LIN {X 0,Y 488.63,Z 370.241,A -85,B 0,C 180,E1 -6427.164,E2 -6427.164} C_VEL
LIN {X 0,Y 488.671,Z 370.238,A -85,B 0,C 180,E1 -6430.331,E2 -6430.331} C_VEL
LIN {X 0,Y 488.668,Z 370.24,A -85,B 0,C 180,E1 -6433.658,E2 -6433.658} C_VEL
LIN {X 0,Y 488.668,Z 370.231,A -85,B 0,C 180,E1 -6436.343,E2 -6436.343} C_VEL
LIN {X 0,Y 488.671,Z 370.225,A -85,B 0,C 180,E1 -6439.67,E2 -6439.67} C_VEL
LIN {X 0,Y 488.65,Z 370.243,A -85,B 0,C 180,E1 -6442.838,E2 -6442.838} C_VEL
LIN {X 0,Y 488.712,Z 370.223,A -85,B 0,C 180,E1 -6445.886,E2 -6445.886} C_VEL
LIN {X 0,Y 488.67,Z 370.24,A -85,B 0,C 180,E1 -6448.819,E2 -6448.819} C_VEL
LIN {X 0,Y 488.695,Z 370.235,A -85,B 0,C 180,E1 -6451.668,E2 -6451.668} C_VEL
LIN {X 0,Y 488.696,Z 370.239,A -85,B 0,C 180,E1 -6454.961,E2 -6454.961} C_VEL
LIN {X 0,Y 488.73,Z 370.261,A -85,B 0,C 180,E1 -6458.266,E2 -6458.266} C_VEL
LIN {X 0,Y 488.873,Z 371.046,A -85,B 0,C 180,E1 -6458.495,E2 -6458.495} C_VEL
LIN {X 0,Y 490.534,Z 379.437,A -85,B 0,C 180,E1 -6460.106,E2 -6460.106} C_VEL
LIN {X 0,Y 490.725,Z 380.846,A -85,B 0,C 180,E1 -6460.313,E2 -6460.313} C_VEL
LIN {X 0,Y 493.718,Z 393.755,A -85,B 0,C 180,E1 -6460.688,E2 -6460.688} C_VEL
LIN {X 0,Y 492.308,Z 519.715,A -85,B 0,C 180,E1 -6462.74,E2 -6462.74} C_VEL
LIN {X 0,Y 492.144,Z 534.173,A -85,B 0,C 180,E1 -6463.145,E2 -6463.145} C_VEL
LIN {X 0,Y 491.844,Z 548.393,A -85,B 0,C 180,E1 -6463.714,E2 -6463.714} C_VEL
LIN {X 0,Y 491.476,Z 562.149,A -85,B 0,C 180,E1 -6464.447,E2 -6464.447} C_VEL
LIN {X 0,Y 491.039,Z 573.092,A -85,B 0,C 180,E1 -6465.177,E2 -6465.177} C_VEL
LIN {X 0,Y 490.649,Z 584.683,A -85,B 0,C 180,E1 -6466.118,E2 -6466.118} C_VEL
LIN {X 0,Y 490.188,Z 595.699,A -85,B 0,C 180,E1 -6467.2,E2 -6467.2} C_VEL
LIN {X 0,Y 489.755,Z 605.882,A -85,B 0,C 180,E1 -6468.41,E2 -6468.41} C_VEL
LIN {X 0,Y 489.407,Z 614.564,A -85,B 0,C 180,E1 -6469.659,E2 -6469.659} C_VEL
LIN {X 0,Y 489.107,Z 622.847,A -85,B 0,C 180,E1 -6471.114,E2 -6471.114} C_VEL
LIN {X 0,Y 488.854,Z 629.502,A -85,B 0,C 180,E1 -6472.566,E2 -6472.566} C_VEL
LIN {X 0,Y 488.751,Z 634.11,A -85,B 0,C 180,E1 -6473.809,E2 -6473.809} C_VEL
LIN {X 0,Y 488.529,Z 637.769,A -85,B 0,C 180,E1 -6475.048,E2 -6475.048} C_VEL
LIN {X 0,Y 488.435,Z 641.375,A -85,B 0,C 180,E1 -6476.7,E2 -6476.7} C_VEL
LIN {X 0,Y 488.484,Z 642.64,A -85,B 0,C 180,E1 -6477.526,E2 -6477.526} C_VEL
LIN {X 0,Y 488.439,Z 644.177,A -85,B 0,C 180,E1 -6479.175,E2 -6479.175} C_VEL
LIN {X 0,Y 488.439,Z 644.37,A -85,B 0,C 180,E1 -6480.824,E2 -6480.824} C_VEL
LIN {X 0,Y 488.495,Z 643.209,A -85,B 0,C 180,E1 -6482.474,E2 -6482.474} C_VEL
LIN {X 0,Y 488.571,Z 640.686,A -85,B 0,C 180,E1 -6484.124,E2 -6484.124} C_VEL
LIN {X 0,Y 488.818,Z 636.708,A -85,B 0,C 180,E1 -6485.776,E2 -6485.776} C_VEL
LIN {X 0,Y 488.963,Z 631.462,A -85,B 0,C 180,E1 -6487.358,E2 -6487.358} C_VEL
LIN {X 0,Y 489.212,Z 625.844,A -85,B 0,C 180,E1 -6488.676,E2 -6488.676} C_VEL
LIN {X 0,Y 489.556,Z 618.17,A -85,B 0,C 180,E1 -6490.129,E2 -6490.129} C_VEL
LIN {X 0,Y 489.943,Z 610.105,A -85,B 0,C 180,E1 -6491.375,E2 -6491.375} C_VEL
LIN {X 0,Y 490.435,Z 600.545,A -85,B 0,C 180,E1 -6492.598,E2 -6492.598} C_VEL
LIN {X 0,Y 490.886,Z 589.425,A -85,B 0,C 180,E1 -6493.77,E2 -6493.77} C_VEL
LIN {X 0,Y 491.245,Z 578.536,A -85,B 0,C 180,E1 -6494.711,E2 -6494.711} C_VEL
LIN {X 0,Y 491.631,Z 566.669,A -85,B 0,C 180,E1 -6495.547,E2 -6495.547} C_VEL
LIN {X 0,Y 492.064,Z 553.581,A -85,B 0,C 180,E1 -6496.278,E2 -6496.278} C_VEL
LIN {X 0,Y 492.329,Z 540.591,A -85,B 0,C 180,E1 -6496.839,E2 -6496.839} C_VEL
LIN {X 0,Y 492.464,Z 526.256,A -85,B 0,C 180,E1 -6497.285,E2 -6497.285} C_VEL
LIN {X 0,Y 492.743,Z 500.215,A -85,B 0,C 180,E1 -6497.777,E2 -6497.777} C_VEL
LIN {X 0,Y 494.504,Z 408.672,A -85,B 0,C 180,E1 -6499.431,E2 -6499.431} C_VEL
LIN {X 0,Y 494.741,Z 394.774,A -85,B 0,C 180,E1 -6499.698,E2 -6499.698} C_VEL
LIN {X 0,Y 492.574,Z 387.053,A -85,B 0,C 180,E1 -6499.998,E2 -6499.998} C_VEL
LIN {X 0,Y 492.44,Z 385.522,A -85,B 0,C 180,E1 -6500.248,E2 -6500.248} C_VEL
LIN {X 0,Y 490.543,Z 377.295,A -85,B 0,C 180,E1 -6502.091,E2 -6502.091} C_VEL
LIN {X 0,Y 488.703,Z 370.295,A -85,B 0,C 180,E1 -6503.773,E2 -6503.773} C_VEL
LIN {X 0,Y 488.797,Z 370.226,A -85,B 0,C 180,E1 -6506.943,E2 -6506.943} C_VEL
LIN {X 0,Y 488.714,Z 370.236,A -85,B 0,C 180,E1 -6510.362,E2 -6510.362} C_VEL
LIN {X 0,Y 488.739,Z 370.23,A -85,B 0,C 180,E1 -6513.484,E2 -6513.484} C_VEL
LIN {X 0,Y 488.678,Z 370.241,A -85,B 0,C 180,E1 -6516.353,E2 -6516.353} C_VEL
LIN {X 0,Y 488.704,Z 370.234,A -85,B 0,C 180,E1 -6519.254,E2 -6519.254} C_VEL
LIN {X 0,Y 488.691,Z 370.24,A -85,B 0,C 180,E1 -6522.525,E2 -6522.525} C_VEL
LIN {X 0,Y 488.705,Z 370.234,A -85,B 0,C 180,E1 -6525.197,E2 -6525.197} C_VEL
LIN {X 0,Y 488.67,Z 370.241,A -85,B 0,C 180,E1 -6528.579,E2 -6528.579} C_VEL
LIN {X 0,Y 488.691,Z 370.237,A -85,B 0,C 180,E1 -6530.949,E2 -6530.949} C_VEL
LIN {X 0,Y 488.648,Z 370.246,A -85,B 0,C 180,E1 -6533.864,E2 -6533.864} C_VEL
LIN {X 0,Y 488.728,Z 370.463,A -85,B 0,C 180,E1 -6536.421,E2 -6536.421} C_VEL
LIN {X 0,Y 491.601,Z 379.515,A -85,B 0,C 180,E1 -6537.795,E2 -6537.795} C_VEL
LIN {X 0,Y 494.839,Z 392.145,A -85,B 0,C 180,E1 -6539.486,E2 -6539.486} C_VEL
LIN {X 0,Y 494.763,Z 398.434,A -85,B 0,C 180,E1 -6540.186,E2 -6540.186} C_VEL
LIN {X 0,Y 493.252,Z 428.365,A -85,B 0,C 180,E1 -6543.331,E2 -6543.331} C_VEL
LIN {X 0,Y 492.07,Z 458.993,A -85,B 0,C 180,E1 -6546.426,E2 -6546.426} C_VEL
LIN {X 0,Y 491.847,Z 465.628,A -85,B 0,C 180,E1 -6547.056,E2 -6547.056} C_VEL
LIN {X 0,Y 494.886,Z 488.681,A -85,B 0,C 180,E1 -6547.594,E2 -6547.594} C_VEL
LIN {X 0,Y 493.486,Z 641.012,A -85,B 0,C 180,E1 -6549.877,E2 -6549.877} C_VEL
LIN {X 0,Y 493.144,Z 656.633,A -85,B 0,C 180,E1 -6550.281,E2 -6550.281} C_VEL
LIN {X 0,Y 492.657,Z 671.656,A -85,B 0,C 180,E1 -6550.845,E2 -6550.845} C_VEL
LIN {X 0,Y 492.069,Z 686.298,A -85,B 0,C 180,E1 -6551.578,E2 -6551.578} C_VEL
LIN {X 0,Y 491.4,Z 699.566,A -85,B 0,C 180,E1 -6552.413,E2 -6552.413} C_VEL
LIN {X 0,Y 490.815,Z 711.781,A -85,B 0,C 180,E1 -6553.357,E2 -6553.357} C_VEL
LIN {X 0,Y 490.13,Z 724.205,A -85,B 0,C 180,E1 -6554.509,E2 -6554.509} C_VEL
LIN {X 0,Y 489.566,Z 736.347,A -85,B 0,C 180,E1 -6555.874,E2 -6555.874} C_VEL
LIN {X 0,Y 489.04,Z 747.102,A -85,B 0,C 180,E1 -6557.339,E2 -6557.339} C_VEL
LIN {X 0,Y 488.679,Z 756.035,A -85,B 0,C 180,E1 -6558.804,E2 -6558.804} C_VEL
LIN {X 0,Y 488.334,Z 764.373,A -85,B 0,C 180,E1 -6560.472,E2 -6560.472} C_VEL
LIN {X 0,Y 488.155,Z 771.047,A -85,B 0,C 180,E1 -6562.138,E2 -6562.138} C_VEL
LIN {X 0,Y 488.079,Z 775.38,A -85,B 0,C 180,E1 -6563.489,E2 -6563.489} C_VEL
LIN {X 0,Y 487.987,Z 779.262,A -85,B 0,C 180,E1 -6565.042,E2 -6565.042} C_VEL
LIN {X 0,Y 488.007,Z 782.201,A -85,B 0,C 180,E1 -6566.696,E2 -6566.696} C_VEL
LIN {X 0,Y 487.941,Z 783.951,A -85,B 0,C 180,E1 -6568.348,E2 -6568.348} C_VEL
LIN {X 0,Y 487.89,Z 784.548,A -85,B 0,C 180,E1 -6569.999,E2 -6569.999} C_VEL
LIN {X 0,Y 487.94,Z 783.95,A -85,B 0,C 180,E1 -6571.649,E2 -6571.649} C_VEL
LIN {X 0,Y 488.012,Z 782.198,A -85,B 0,C 180,E1 -6573.301,E2 -6573.301} C_VEL
LIN {X 0,Y 487.981,Z 779.264,A -85,B 0,C 180,E1 -6574.956,E2 -6574.956} C_VEL
LIN {X 0,Y 488.038,Z 775.078,A -85,B 0,C 180,E1 -6576.614,E2 -6576.614} C_VEL
LIN {X 0,Y 488.197,Z 769.522,A -85,B 0,C 180,E1 -6578.276,E2 -6578.276} C_VEL
LIN {X 0,Y 488.368,Z 762.446,A -85,B 0,C 180,E1 -6579.943,E2 -6579.943} C_VEL
LIN {X 0,Y 488.711,Z 754.857,A -85,B 0,C 180,E1 -6581.403,E2 -6581.403} C_VEL
LIN {X 0,Y 489.079,Z 745.703,A -85,B 0,C 180,E1 -6582.868,E2 -6582.868} C_VEL
LIN {X 0,Y 489.529,Z 736.367,A -85,B 0,C 180,E1 -6584.125,E2 -6584.125} C_VEL
LIN {X 0,Y 490.102,Z 724.237,A -85,B 0,C 180,E1 -6585.489,E2 -6585.489} C_VEL
LIN {X 0,Y 490.84,Z 711.822,A -85,B 0,C 180,E1 -6586.639,E2 -6586.639} C_VEL
LIN {X 0,Y 491.394,Z 699.601,A -85,B 0,C 180,E1 -6587.584,E2 -6587.584} C_VEL
LIN {X 0,Y 491.997,Z 686.334,A -85,B 0,C 180,E1 -6588.422,E2 -6588.422} C_VEL
LIN {X 0,Y 492.632,Z 671.724,A -85,B 0,C 180,E1 -6589.153,E2 -6589.153} C_VEL
LIN {X 0,Y 493.115,Z 656.455,A -85,B 0,C 180,E1 -6589.727,E2 -6589.727} C_VEL
LIN {X 0,Y 493.476,Z 641.155,A -85,B 0,C 180,E1 -6590.121,E2 -6590.121} C_VEL
LIN {X 0,Y 494.854,Z 499.188,A -85,B 0,C 180,E1 -6592.285,E2 -6592.285} C_VEL
LIN {X 0,Y 494.849,Z 487.544,A -85,B 0,C 180,E1 -6592.477,E2 -6592.477} C_VEL
LIN {X 0,Y 492.247,Z 468.47,A -85,B 0,C 180,E1 -6592.933,E2 -6592.933} C_VEL
LIN {X 0,Y 493.504,Z 436.983,A -85,B 0,C 180,E1 -6596.083,E2 -6596.083} C_VEL
LIN {X 0,Y 494.721,Z 409.612,A -85,B 0,C 180,E1 -6598.88,E2 -6598.88} C_VEL
LIN {X 0,Y 495.442,Z 394.035,A -85,B 0,C 180,E1 -6600.497,E2 -6600.497} C_VEL
LIN {X 0,Y 491.474,Z 379.619,A -85,B 0,C 180,E1 -6602.288,E2 -6602.288} C_VEL
LIN {X 0,Y 488.735,Z 370.407,A -85,B 0,C 180,E1 -6603.512,E2 -6603.512} C_VEL
LIN {X 0,Y 488.639,Z 370.245,A -85,B 0,C 180,E1 -6606.348,E2 -6606.348} C_VEL
LIN {X 0,Y 488.676,Z 370.237,A -85,B 0,C 180,E1 -6609.254,E2 -6609.254} C_VEL
LIN {X 0,Y 488.655,Z 370.244,A -85,B 0,C 180,E1 -6612.527,E2 -6612.527} C_VEL
LIN {X 0,Y 488.685,Z 370.234,A -85,B 0,C 180,E1 -6615.196,E2 -6615.196} C_VEL
LIN {X 0,Y 488.647,Z 370.228,A -85,B 0,C 180,E1 -6618.578,E2 -6618.578} C_VEL
LIN {X 0,Y 488.674,Z 370.237,A -85,B 0,C 180,E1 -6620.949,E2 -6620.949} C_VEL
LIN {X 0,Y 488.631,Z 370.228,A -85,B 0,C 180,E1 -6623.864,E2 -6623.864} C_VEL
LIN {X 0,Y 488.695,Z 370.226,A -85,B 0,C 180,E1 -6626.519,E2 -6626.519} C_VEL
LIN {X 0,Y 488.703,Z 370.232,A -85,B 0,C 180,E1 -6629.779,E2 -6629.779} C_VEL
LIN {X 0,Y 488.684,Z 370.234,A -85,B 0,C 180,E1 -6633.077,E2 -6633.077} C_VEL
LIN {X 0,Y 488.653,Z 370.236,A -85,B 0,C 180,E1 -6636.253,E2 -6636.253} C_VEL
LIN {X 0,Y 488.731,Z 370.223,A -85,B 0,C 180,E1 -6639.175,E2 -6639.175} C_VEL
LIN {X 0,Y 488.73,Z 370.226,A -85,B 0,C 180,E1 -6641.632,E2 -6641.632} C_VEL
LIN {X 0,Y 488.73,Z 370.223,A -85,B 0,C 180,E1 -6644.999,E2 -6644.999} C_VEL
LIN {X 0,Y 488.787,Z 370.228,A -85,B 0,C 180,E1 -6648.387,E2 -6648.387} C_VEL
LIN {X 0,Y 488.741,Z 370.223,A -85,B 0,C 180,E1 -6651.732,E2 -6651.732} C_VEL
LIN {X 0,Y 488.787,Z 370.224,A -85,B 0,C 180,E1 -6654.224,E2 -6654.224} C_VEL
LIN {X 0,Y 488.93,Z 370.201,A -85,B 0,C 180,E1 -6657.529,E2 -6657.529} C_VEL
LIN {X 0,Y 488.895,Z 370.203,A -85,B 0,C 180,E1 -6660.824,E2 -6660.824} C_VEL
LIN {X 0,Y 488.929,Z 370.203,A -85,B 0,C 180,E1 -6662.472,E2 -6662.472} C_VEL
LIN {X 0,Y 488.817,Z 370.213,A -85,B 0,C 180,E1 -6665.776,E2 -6665.776} C_VEL
LIN {X 0,Y 488.757,Z 370.224,A -85,B 0,C 180,E1 -6668.267,E2 -6668.267} C_VEL
LIN {X 0,Y 488.787,Z 370.212,A -85,B 0,C 180,E1 -6671.613,E2 -6671.613} C_VEL
LIN {X 0,Y 488.74,Z 370.226,A -85,B 0,C 180,E1 -6675.001,E2 -6675.001} C_VEL
LIN {X 0,Y 488.73,Z 370.23,A -85,B 0,C 180,E1 -6678.443,E2 -6678.443} C_VEL
LIN {X 0,Y 488.692,Z 370.23,A -85,B 0,C 180,E1 -6681.072,E2 -6681.072} C_VEL
LIN {X 0,Y 488.653,Z 370.237,A -85,B 0,C 180,E1 -6683.748,E2 -6683.748} C_VEL
LIN {X 0,Y 488.681,Z 370.24,A -85,B 0,C 180,E1 -6686.922,E2 -6686.922} C_VEL
LIN {X 0,Y 488.683,Z 370.234,A -85,B 0,C 180,E1 -6690.222,E2 -6690.222} C_VEL
LIN {X 0,Y 488.697,Z 370.234,A -85,B 0,C 180,E1 -6693.481,E2 -6693.481} C_VEL
LIN {X 0,Y 488.655,Z 370.235,A -85,B 0,C 180,E1 -6696.353,E2 -6696.353} C_VEL
LIN {X 0,Y 488.674,Z 370.238,A -85,B 0,C 180,E1 -6699.257,E2 -6699.257} C_VEL
LIN {X 0,Y 488.654,Z 370.232,A -85,B 0,C 180,E1 -6701.596,E2 -6701.596} C_VEL
LIN {X 0,Y 488.684,Z 370.242,A -85,B 0,C 180,E1 -6704.805,E2 -6704.805} C_VEL
LIN {X 0,Y 488.637,Z 370.24,A -85,B 0,C 180,E1 -6707.471,E2 -6707.471} C_VEL
LIN {X 0,Y 488.694,Z 370.229,A -85,B 0,C 180,E1 -6709.675,E2 -6709.675} C_VEL
LIN {X 0,Y 488.641,Z 370.237,A -85,B 0,C 180,E1 -6712.84,E2 -6712.84} C_VEL
LIN {X 0,Y 488.726,Z 370.405,A -85,B 0,C 180,E1 -6715.64,E2 -6715.64} C_VEL
LIN {X 0,Y 494.002,Z 388.467,A -85,B 0,C 180,E1 -6718.007,E2 -6718.007} C_VEL
LIN {X 0,Y 495.447,Z 393.988,A -85,B 0,C 180,E1 -6718.704,E2 -6718.704} C_VEL
LIN {X 0,Y 494.7,Z 414.108,A -85,B 0,C 180,E1 -6720.883,E2 -6720.883} C_VEL
LIN {X 0,Y 493.899,Z 418.535,A -85,B 0,C 180,E1 -6721.327,E2 -6721.327} C_VEL
LIN {X 0,Y 487.94,Z 433.643,A -85,B 0,C 180,E1 -6722.661,E2 -6722.661} C_VEL
LIN {X 0,Y 487.139,Z 438.124,A -85,B 0,C 180,E1 -6723.107,E2 -6723.107} C_VEL
LIN {X 0,Y 486.163,Z 465.721,A -85,B 0,C 180,E1 -6726.003,E2 -6726.003} C_VEL
LIN {X 0,Y 486.002,Z 472.632,A -85,B 0,C 180,E1 -6726.667,E2 -6726.667} C_VEL
LIN {X 0,Y 489.058,Z 491.11,A -85,B 0,C 180,E1 -6727.121,E2 -6727.121} C_VEL
LIN {X 0,Y 487.462,Z 640.161,A -85,B 0,C 180,E1 -6729.386,E2 -6729.386} C_VEL
LIN {X 0,Y 487.095,Z 655.841,A -85,B 0,C 180,E1 -6729.784,E2 -6729.784} C_VEL
LIN {X 0,Y 486.549,Z 669.962,A -85,B 0,C 180,E1 -6730.3,E2 -6730.3} C_VEL
LIN {X 0,Y 485.868,Z 684.559,A -85,B 0,C 180,E1 -6731.008,E2 -6731.008} C_VEL
LIN {X 0,Y 485.181,Z 698.293,A -85,B 0,C 180,E1 -6731.856,E2 -6731.856} C_VEL
LIN {X 0,Y 484.446,Z 710.916,A -85,B 0,C 180,E1 -6732.809,E2 -6732.809} C_VEL
LIN {X 0,Y 483.726,Z 723.662,A -85,B 0,C 180,E1 -6733.977,E2 -6733.977} C_VEL
LIN {X 0,Y 483.079,Z 733.473,A -85,B 0,C 180,E1 -6735.036,E2 -6735.036} C_VEL
LIN {X 0,Y 482.501,Z 743.486,A -85,B 0,C 180,E1 -6736.31,E2 -6736.31} C_VEL
LIN {X 0,Y 481.985,Z 753.507,A -85,B 0,C 180,E1 -6737.835,E2 -6737.835} C_VEL
LIN {X 0,Y 481.598,Z 761.397,A -85,B 0,C 180,E1 -6739.278,E2 -6739.278} C_VEL
LIN {X 0,Y 481.241,Z 768.131,A -85,B 0,C 180,E1 -6740.757,E2 -6740.757} C_VEL
LIN {X 0,Y 481.014,Z 774.375,A -85,B 0,C 180,E1 -6742.445,E2 -6742.445} C_VEL
LIN {X 0,Y 480.917,Z 779.203,A -85,B 0,C 180,E1 -6744.13,E2 -6744.13} C_VEL
LIN {X 0,Y 480.796,Z 782.742,A -85,B 0,C 180,E1 -6745.81,E2 -6745.81} C_VEL
LIN {X 0,Y 480.799,Z 785.083,A -85,B 0,C 180,E1 -6747.488,E2 -6747.488} C_VEL
LIN {X 0,Y 480.757,Z 786.278,A -85,B 0,C 180,E1 -6749.164,E2 -6749.164} C_VEL
LIN {X 0,Y 480.757,Z 786.295,A -85,B 0,C 180,E1 -6750.839,E2 -6750.839} C_VEL
LIN {X 0,Y 480.8,Z 785.169,A -85,B 0,C 180,E1 -6752.515,E2 -6752.515} C_VEL
LIN {X 0,Y 480.796,Z 782.895,A -85,B 0,C 180,E1 -6754.193,E2 -6754.193} C_VEL
LIN {X 0,Y 480.9,Z 779.42,A -85,B 0,C 180,E1 -6755.873,E2 -6755.873} C_VEL
LIN {X 0,Y 481.01,Z 774.663,A -85,B 0,C 180,E1 -6757.557,E2 -6757.557} C_VEL
LIN {X 0,Y 481.226,Z 768.503,A -85,B 0,C 180,E1 -6759.246,E2 -6759.246} C_VEL
LIN {X 0,Y 481.629,Z 760.754,A -85,B 0,C 180,E1 -6760.936,E2 -6760.936} C_VEL
LIN {X 0,Y 482.003,Z 752.225,A -85,B 0,C 180,E1 -6762.463,E2 -6762.463} C_VEL
LIN {X 0,Y 482.569,Z 742.54,A -85,B 0,C 180,E1 -6763.905,E2 -6763.905} C_VEL
LIN {X 0,Y 483.144,Z 732.385,A -85,B 0,C 180,E1 -6765.18,E2 -6765.18} C_VEL
LIN {X 0,Y 483.874,Z 720.993,A -85,B 0,C 180,E1 -6766.381,E2 -6766.381} C_VEL
LIN {X 0,Y 484.608,Z 708.092,A -85,B 0,C 180,E1 -6767.514,E2 -6767.514} C_VEL
LIN {X 0,Y 485.393,Z 694.88,A -85,B 0,C 180,E1 -6768.466,E2 -6768.466} C_VEL
LIN {X 0,Y 486.061,Z 681.287,A -85,B 0,C 180,E1 -6769.261,E2 -6769.261} C_VEL
LIN {X 0,Y 486.681,Z 666.702,A -85,B 0,C 180,E1 -6769.927,E2 -6769.927} C_VEL
LIN {X 0,Y 487.203,Z 651.649,A -85,B 0,C 180,E1 -6770.435,E2 -6770.435} C_VEL
LIN {X 0,Y 487.565,Z 635.65,A -85,B 0,C 180,E1 -6770.789,E2 -6770.789} C_VEL
LIN {X 0,Y 489.071,Z 490.942,A -85,B 0,C 180,E1 -6772.972,E2 -6772.972} C_VEL
LIN {X 0,Y 485.975,Z 472.205,A -85,B 0,C 180,E1 -6773.448,E2 -6773.448} C_VEL
LIN {X 0,Y 486.713,Z 448.579,A -85,B 0,C 180,E1 -6775.872,E2 -6775.872} C_VEL
LIN {X 0,Y 487.808,Z 421.261,A -85,B 0,C 180,E1 -6778.812,E2 -6778.812} C_VEL
LIN {X 0,Y 488.856,Z 396.737,A -85,B 0,C 180,E1 -6781.487,E2 -6781.487} C_VEL
LIN {X 0,Y 485.329,Z 383.414,A -85,B 0,C 180,E1 -6783.202,E2 -6783.202} C_VEL
LIN {X 0,Y 481.629,Z 371.34,A -85,B 0,C 180,E1 -6784.829,E2 -6784.829} C_VEL
LIN {X 0,Y 481.587,Z 371.116,A -85,B 0,C 180,E1 -6786.617,E2 -6786.617} C_VEL
LIN {X 0,Y 481.632,Z 371.111,A -85,B 0,C 180,E1 -6789.342,E2 -6789.342} C_VEL
LIN {X 0,Y 481.612,Z 371.107,A -85,B 0,C 180,E1 -6792.166,E2 -6792.166} C_VEL
LIN {X 0,Y 481.654,Z 371.112,A -85,B 0,C 180,E1 -6794.459,E2 -6794.459} C_VEL
LIN {X 0,Y 481.612,Z 371.117,A -85,B 0,C 180,E1 -6797.835,E2 -6797.835} C_VEL
LIN {X 0,Y 481.625,Z 371.11,A -85,B 0,C 180,E1 -6801.136,E2 -6801.136} C_VEL
LIN {X 0,Y 481.618,Z 371.108,A -85,B 0,C 180,E1 -6804.289,E2 -6804.289} C_VEL
LIN {X 0,Y 481.675,Z 371.099,A -85,B 0,C 180,E1 -6806.327,E2 -6806.327} C_VEL
LIN {X 0,Y 481.631,Z 371.118,A -85,B 0,C 180,E1 -6809.423,E2 -6809.423} C_VEL
LIN {X 0,Y 481.649,Z 371.111,A -85,B 0,C 180,E1 -6812.165,E2 -6812.165} C_VEL
LIN {X 0,Y 481.67,Z 371.114,A -85,B 0,C 180,E1 -6814.967,E2 -6814.967} C_VEL
LIN {X 0,Y 481.708,Z 371.32,A -85,B 0,C 180,E1 -6818.13,E2 -6818.13} C_VEL
LIN {X 0,Y 483.601,Z 380.575,A -85,B 0,C 180,E1 -6819.919,E2 -6819.919} C_VEL
LIN {X 0,Y 483.905,Z 381.906,A -85,B 0,C 180,E1 -6820.05,E2 -6820.05} C_VEL
LIN {X 0,Y 486.909,Z 394.286,A -85,B 0,C 180,E1 -6820.41,E2 -6820.41} C_VEL
LIN {X 0,Y 485.9,Z 484.424,A -85,B 0,C 180,E1 -6821.909,E2 -6821.909} C_VEL
LIN {X 0,Y 485.496,Z 520.889,A -85,B 0,C 180,E1 -6822.528,E2 -6822.528} C_VEL
LIN {X 0,Y 485.33,Z 535.642,A -85,B 0,C 180,E1 -6822.955,E2 -6822.955} C_VEL
LIN {X 0,Y 485.008,Z 549.682,A -85,B 0,C 180,E1 -6823.532,E2 -6823.532} C_VEL
LIN {X 0,Y 484.641,Z 562.452,A -85,B 0,C 180,E1 -6824.222,E2 -6824.222} C_VEL
LIN {X 0,Y 484.2,Z 573.506,A -85,B 0,C 180,E1 -6824.963,E2 -6824.963} C_VEL
LIN {X 0,Y 483.779,Z 585.19,A -85,B 0,C 180,E1 -6825.917,E2 -6825.917} C_VEL
LIN {X 0,Y 483.275,Z 596.818,A -85,B 0,C 180,E1 -6827.071,E2 -6827.071} C_VEL
LIN {X 0,Y 482.838,Z 606.54,A -85,B 0,C 180,E1 -6828.242,E2 -6828.242} C_VEL
LIN {X 0,Y 482.462,Z 615.289,A -85,B 0,C 180,E1 -6829.509,E2 -6829.509} C_VEL
LIN {X 0,Y 482.127,Z 623.647,A -85,B 0,C 180,E1 -6830.984,E2 -6830.984} C_VEL
LIN {X 0,Y 481.875,Z 630.351,A -85,B 0,C 180,E1 -6832.457,E2 -6832.457} C_VEL
LIN {X 0,Y 481.76,Z 634.996,A -85,B 0,C 180,E1 -6833.719,E2 -6833.719} C_VEL
LIN {X 0,Y 481.496,Z 639.77,A -85,B 0,C 180,E1 -6835.395,E2 -6835.395} C_VEL
LIN {X 0,Y 481.412,Z 642.347,A -85,B 0,C 180,E1 -6836.652,E2 -6836.652} C_VEL
LIN {X 0,Y 481.471,Z 643.628,A -85,B 0,C 180,E1 -6837.49,E2 -6837.49} C_VEL
LIN {X 0,Y 481.426,Z 645.196,A -85,B 0,C 180,E1 -6839.163,E2 -6839.163} C_VEL
LIN {X 0,Y 481.427,Z 645.413,A -85,B 0,C 180,E1 -6840.836,E2 -6840.836} C_VEL
LIN {X 0,Y 481.486,Z 644.266,A -85,B 0,C 180,E1 -6842.51,E2 -6842.51} C_VEL
LIN {X 0,Y 481.567,Z 641.75,A -85,B 0,C 180,E1 -6844.185,E2 -6844.185} C_VEL
LIN {X 0,Y 481.836,Z 637.77,A -85,B 0,C 180,E1 -6845.86,E2 -6845.86} C_VEL
LIN {X 0,Y 481.995,Z 632.523,A -85,B 0,C 180,E1 -6847.467,E2 -6847.467} C_VEL
LIN {X 0,Y 482.27,Z 626.922,A -85,B 0,C 180,E1 -6848.802,E2 -6848.802} C_VEL
LIN {X 0,Y 482.66,Z 619.262,A -85,B 0,C 180,E1 -6850.275,E2 -6850.275} C_VEL
LIN {X 0,Y 483.085,Z 611.189,A -85,B 0,C 180,E1 -6851.539,E2 -6851.539} C_VEL
LIN {X 0,Y 483.581,Z 601.61,A -85,B 0,C 180,E1 -6852.779,E2 -6852.779} C_VEL
LIN {X 0,Y 484.07,Z 590.454,A -85,B 0,C 180,E1 -6853.967,E2 -6853.967} C_VEL
LIN {X 0,Y 484.462,Z 579.527,A -85,B 0,C 180,E1 -6854.921,E2 -6854.921} C_VEL
LIN {X 0,Y 484.862,Z 567.644,A -85,B 0,C 180,E1 -6855.77,E2 -6855.77} C_VEL
LIN {X 0,Y 485.339,Z 554.6,A -85,B 0,C 180,E1 -6856.51,E2 -6856.51} C_VEL
LIN {X 0,Y 485.61,Z 542.435,A -85,B 0,C 180,E1 -6857.051,E2 -6857.051} C_VEL
LIN {X 0,Y 485.715,Z 528.411,A -85,B 0,C 180,E1 -6857.51,E2 -6857.51} C_VEL
LIN {X 0,Y 485.959,Z 507.762,A -85,B 0,C 180,E1 -6857.925,E2 -6857.925} C_VEL
LIN {X 0,Y 487.743,Z 420.488,A -85,B 0,C 180,E1 -6859.546,E2 -6859.546} C_VEL
LIN {X 0,Y 488.183,Z 395.696,A -85,B 0,C 180,E1 -6860.039,E2 -6860.039} C_VEL
LIN {X 0,Y 485.964,Z 388.277,A -85,B 0,C 180,E1 -6860.344,E2 -6860.344} C_VEL
LIN {X 0,Y 485.648,Z 387.025,A -85,B 0,C 180,E1 -6860.544,E2 -6860.544} C_VEL
LIN {X 0,Y 483.703,Z 378.84,A -85,B 0,C 180,E1 -6862.42,E2 -6862.42} C_VEL
LIN {X 0,Y 481.715,Z 371.165,A -85,B 0,C 180,E1 -6864.312,E2 -6864.312} C_VEL
LIN {X 0,Y 481.751,Z 371.104,A -85,B 0,C 180,E1 -6867.139,E2 -6867.139} C_VEL
LIN {X 0,Y 481.684,Z 371.11,A -85,B 0,C 180,E1 -6869.741,E2 -6869.741} C_VEL
LIN {X 0,Y 481.677,Z 371.113,A -85,B 0,C 180,E1 -6872.674,E2 -6872.674} C_VEL
LIN {X 0,Y 481.665,Z 371.112,A -85,B 0,C 180,E1 -6875.203,E2 -6875.203} C_VEL
LIN {X 0,Y 481.674,Z 371.112,A -85,B 0,C 180,E1 -6878.859,E2 -6878.859} C_VEL
LIN {X 0,Y 481.65,Z 371.116,A -85,B 0,C 180,E1 -6881.911,E2 -6881.911} C_VEL
LIN {X 0,Y 481.658,Z 371.116,A -85,B 0,C 180,E1 -6884.457,E2 -6884.457} C_VEL
LIN {X 0,Y 481.628,Z 371.119,A -85,B 0,C 180,E1 -6887.836,E2 -6887.836} C_VEL
LIN {X 0,Y 481.652,Z 371.115,A -85,B 0,C 180,E1 -6890.655,E2 -6890.655} C_VEL
LIN {X 0,Y 481.609,Z 371.119,A -85,B 0,C 180,E1 -6893.379,E2 -6893.379} C_VEL
LIN {X 0,Y 481.708,Z 371.307,A -85,B 0,C 180,E1 -6895.905,E2 -6895.905} C_VEL
LIN {X 0,Y 485.064,Z 381.911,A -85,B 0,C 180,E1 -6897.581,E2 -6897.581} C_VEL
LIN {X 0,Y 488.184,Z 394.044,A -85,B 0,C 180,E1 -6899.265,E2 -6899.265} C_VEL
LIN {X 0,Y 488.26,Z 398.178,A -85,B 0,C 180,E1 -6899.748,E2 -6899.748} C_VEL
LIN {X 0,Y 486.737,Z 424.588,A -85,B 0,C 180,E1 -6902.596,E2 -6902.596} C_VEL
LIN {X 0,Y 485.382,Z 455.536,A -85,B 0,C 180,E1 -6905.811,E2 -6905.811} C_VEL
LIN {X 0,Y 485.056,Z 464.405,A -85,B 0,C 180,E1 -6906.687,E2 -6906.687} C_VEL
LIN {X 0,Y 486.937,Z 479.661,A -85,B 0,C 180,E1 -6907.064,E2 -6907.064} C_VEL
LIN {X 0,Y 488.303,Z 490.714,A -85,B 0,C 180,E1 -6907.304,E2 -6907.304} C_VEL
LIN {X 0,Y 486.839,Z 641.179,A -85,B 0,C 180,E1 -6909.59,E2 -6909.59} C_VEL
LIN {X 0,Y 486.468,Z 656.504,A -85,B 0,C 180,E1 -6909.991,E2 -6909.991} C_VEL
LIN {X 0,Y 485.957,Z 671.728,A -85,B 0,C 180,E1 -6910.57,E2 -6910.57} C_VEL
LIN {X 0,Y 485.293,Z 686.354,A -85,B 0,C 180,E1 -6911.311,E2 -6911.311} C_VEL
LIN {X 0,Y 484.633,Z 699.612,A -85,B 0,C 180,E1 -6912.16,E2 -6912.16} C_VEL
LIN {X 0,Y 483.922,Z 712.988,A -85,B 0,C 180,E1 -6913.215,E2 -6913.215} C_VEL
LIN {X 0,Y 483.179,Z 725.264,A -85,B 0,C 180,E1 -6914.389,E2 -6914.389} C_VEL
LIN {X 0,Y 482.628,Z 736.375,A -85,B 0,C 180,E1 -6915.666,E2 -6915.666} C_VEL
LIN {X 0,Y 482.051,Z 747.126,A -85,B 0,C 180,E1 -6917.153,E2 -6917.153} C_VEL
LIN {X 0,Y 481.67,Z 756.056,A -85,B 0,C 180,E1 -6918.639,E2 -6918.639} C_VEL
LIN {X 0,Y 481.27,Z 764.392,A -85,B 0,C 180,E1 -6920.331,E2 -6920.331} C_VEL
LIN {X 0,Y 481.105,Z 771.064,A -85,B 0,C 180,E1 -6922.022,E2 -6922.022} C_VEL
LIN {X 0,Y 481.007,Z 775.675,A -85,B 0,C 180,E1 -6923.488,E2 -6923.488} C_VEL
LIN {X 0,Y 480.913,Z 779.277,A -85,B 0,C 180,E1 -6924.968,E2 -6924.968} C_VEL
LIN {X 0,Y 480.931,Z 782.215,A -85,B 0,C 180,E1 -6926.648,E2 -6926.648} C_VEL
LIN {X 0,Y 480.869,Z 783.965,A -85,B 0,C 180,E1 -6928.324,E2 -6928.324} C_VEL
LIN {X 0,Y 480.809,Z 784.562,A -85,B 0,C 180,E1 -6929.999,E2 -6929.999} C_VEL
LIN {X 0,Y 480.868,Z 783.964,A -85,B 0,C 180,E1 -6931.674,E2 -6931.674} C_VEL
LIN {X 0,Y 480.934,Z 782.213,A -85,B 0,C 180,E1 -6933.35,E2 -6933.35} C_VEL
LIN {X 0,Y 480.906,Z 779.28,A -85,B 0,C 180,E1 -6935.029,E2 -6935.029} C_VEL
LIN {X 0,Y 480.958,Z 775.094,A -85,B 0,C 180,E1 -6936.712,E2 -6936.712} C_VEL
LIN {X 0,Y 481.113,Z 769.539,A -85,B 0,C 180,E1 -6938.398,E2 -6938.398} C_VEL
LIN {X 0,Y 481.326,Z 762.465,A -85,B 0,C 180,E1 -6940.09,E2 -6940.09} C_VEL
LIN {X 0,Y 481.667,Z 754.879,A -85,B 0,C 180,E1 -6941.572,E2 -6941.572} C_VEL
LIN {X 0,Y 482.091,Z 745.728,A -85,B 0,C 180,E1 -6943.058,E2 -6943.058} C_VEL
LIN {X 0,Y 482.587,Z 736.394,A -85,B 0,C 180,E1 -6944.332,E2 -6944.332} C_VEL
LIN {X 0,Y 483.154,Z 725.293,A -85,B 0,C 180,E1 -6945.609,E2 -6945.609} C_VEL
LIN {X 0,Y 483.946,Z 713.078,A -85,B 0,C 180,E1 -6946.777,E2 -6946.777} C_VEL
LIN {X 0,Y 484.609,Z 699.647,A -85,B 0,C 180,E1 -6947.839,E2 -6947.839} C_VEL
LIN {X 0,Y 485.244,Z 686.389,A -85,B 0,C 180,E1 -6948.688,E2 -6948.688} C_VEL
LIN {X 0,Y 485.928,Z 671.793,A -85,B 0,C 180,E1 -6949.428,E2 -6949.428} C_VEL
LIN {X 0,Y 486.442,Z 656.797,A -85,B 0,C 180,E1 -6950.001,E2 -6950.001} C_VEL
LIN {X 0,Y 486.828,Z 641.309,A -85,B 0,C 180,E1 -6950.408,E2 -6950.408} C_VEL
LIN {X 0,Y 488.314,Z 489.212,A -85,B 0,C 180,E1 -6952.738,E2 -6952.738} C_VEL
LIN {X 0,Y 485.405,Z 467.989,A -85,B 0,C 180,E1 -6953.25,E2 -6953.25} C_VEL
LIN {X 0,Y 486.751,Z 437.596,A -85,B 0,C 180,E1 -6956.331,E2 -6956.331} C_VEL
LIN {X 0,Y 488.037,Z 409.988,A -85,B 0,C 180,E1 -6959.195,E2 -6959.195} C_VEL
LIN {X 0,Y 488.699,Z 395.715,A -85,B 0,C 180,E1 -6960.696,E2 -6960.696} C_VEL
LIN {X 0,Y 483.657,Z 377.985,A -85,B 0,C 180,E1 -6962.949,E2 -6962.949} C_VEL
LIN {X 0,Y 481.692,Z 371.271,A -85,B 0,C 180,E1 -6963.868,E2 -6963.868} C_VEL
LIN {X 0,Y 481.595,Z 371.12,A -85,B 0,C 180,E1 -6966.747,E2 -6966.747} C_VEL
LIN {X 0,Y 481.644,Z 371.116,A -85,B 0,C 180,E1 -6969.941,E2 -6969.941} C_VEL
LIN {X 0,Y 481.61,Z 371.115,A -85,B 0,C 180,E1 -6973.301,E2 -6973.301} C_VEL
LIN {X 0,Y 481.636,Z 371.113,A -85,B 0,C 180,E1 -6975.641,E2 -6975.641} C_VEL
LIN {X 0,Y 481.609,Z 371.11,A -85,B 0,C 180,E1 -6978.953,E2 -6978.953} C_VEL
LIN {X 0,Y 481.616,Z 371.118,A -85,B 0,C 180,E1 -6981.996,E2 -6981.996} C_VEL
LIN {X 0,Y 481.664,Z 371.089,A -85,B 0,C 180,E1 -6985.316,E2 -6985.316} C_VEL
LIN {X 0,Y 481.627,Z 371.118,A -85,B 0,C 180,E1 -6988.31,E2 -6988.31} C_VEL
LIN {X 0,Y 481.644,Z 371.107,A -85,B 0,C 180,E1 -6991.215,E2 -6991.215} C_VEL
LIN {X 0,Y 481.63,Z 371.115,A -85,B 0,C 180,E1 -6994.039,E2 -6994.039} C_VEL
LIN {X 0,Y 481.638,Z 371.115,A -85,B 0,C 180,E1 -6996.817,E2 -6996.817} C_VEL
LIN {X 0,Y 481.676,Z 371.101,A -85,B 0,C 180,E1 -6999.502,E2 -6999.502} C_VEL
LIN {X 0,Y 481.652,Z 371.112,A -85,B 0,C 180,E1 -7002.156,E2 -7002.156} C_VEL
LIN {X 0,Y 481.712,Z 371.098,A -85,B 0,C 180,E1 -7004.775,E2 -7004.775} C_VEL
LIN {X 0,Y 481.733,Z 371.104,A -85,B 0,C 180,E1 -7008.215,E2 -7008.215} C_VEL
LIN {X 0,Y 481.7,Z 371.099,A -85,B 0,C 180,E1 -7011.611,E2 -7011.611} C_VEL
LIN {X 0,Y 481.748,Z 371.1,A -85,B 0,C 180,E1 -7014.139,E2 -7014.139} C_VEL
LIN {X 0,Y 481.897,Z 371.077,A -85,B 0,C 180,E1 -7017.492,E2 -7017.492} C_VEL
LIN {X 0,Y 481.848,Z 371.08,A -85,B 0,C 180,E1 -7020.836,E2 -7020.836} C_VEL
LIN {X 0,Y 481.895,Z 371.079,A -85,B 0,C 180,E1 -7022.508,E2 -7022.508} C_VEL
LIN {X 0,Y 481.777,Z 371.091,A -85,B 0,C 180,E1 -7025.861,E2 -7025.861} C_VEL
LIN {X 0,Y 481.712,Z 371.103,A -85,B 0,C 180,E1 -7028.389,E2 -7028.389} C_VEL
LIN {X 0,Y 481.733,Z 371.09,A -85,B 0,C 180,E1 -7031.785,E2 -7031.785} C_VEL
LIN {X 0,Y 481.723,Z 371.098,A -85,B 0,C 180,E1 -7035.225,E2 -7035.225} C_VEL
LIN {X 0,Y 481.692,Z 371.111,A -85,B 0,C 180,E1 -7038.723,E2 -7038.723} C_VEL
LIN {X 0,Y 481.63,Z 371.108,A -85,B 0,C 180,E1 -7041.396,E2 -7041.396} C_VEL
LIN {X 0,Y 481.632,Z 371.114,A -85,B 0,C 180,E1 -7044.116,E2 -7044.116} C_VEL
LIN {X 0,Y 481.636,Z 371.115,A -85,B 0,C 180,E1 -7047.118,E2 -7047.118} C_VEL
LIN {X 0,Y 481.637,Z 371.109,A -85,B 0,C 180,E1 -7049.744,E2 -7049.744} C_VEL
LIN {X 0,Y 481.635,Z 371.115,A -85,B 0,C 180,E1 -7052.677,E2 -7052.677} C_VEL
LIN {X 0,Y 481.616,Z 371.113,A -85,B 0,C 180,E1 -7055.711,E2 -7055.711} C_VEL
LIN {X 0,Y 481.618,Z 371.111,A -85,B 0,C 180,E1 -7058.864,E2 -7058.864} C_VEL
LIN {X 0,Y 481.608,Z 371.109,A -85,B 0,C 180,E1 -7061.91,E2 -7061.91} C_VEL
LIN {X 0,Y 481.638,Z 371.115,A -85,B 0,C 180,E1 -7064.46,E2 -7064.46} C_VEL
LIN {X 0,Y 481.601,Z 371.111,A -85,B 0,C 180,E1 -7066.857,E2 -7066.857} C_VEL
LIN {X 0,Y 481.645,Z 371.106,A -85,B 0,C 180,E1 -7070.059,E2 -7070.059} C_VEL
LIN {X 0,Y 481.599,Z 371.114,A -85,B 0,C 180,E1 -7073.381,E2 -7073.381} C_VEL
LIN {X 0,Y 481.678,Z 371.192,A -85,B 0,C 180,E1 -7075.223,E2 -7075.223} C_VEL
LIN {X 0,Y 481.976,Z 372.457,A -85,B 0,C 180,E1 -7075.447,E2 -7075.447} C_VEL
LIN {X 0,Y 486.926,Z 389.013,A -85,B 0,C 180,E1 -7077.626,E2 -7077.626} C_VEL
LIN {X 0,Y 488.808,Z 396.09,A -85,B 0,C 180,E1 -7078.531,E2 -7078.531} C_VEL
LIN {X 0,Y 487.944,Z 416.867,A -85,B 0,C 180,E1 -7080.799,E2 -7080.799} C_VEL
LIN {X 0,Y 487.139,Z 438.124,A -85,B 0,C 180,E1 -7083.107,E2 -7083.107} C_VEL
LIN {X 0,Y 486.343,Z 442.609,A -85,B 0,C 180,E1 -7083.55,E2 -7083.55} C_VEL
LIN {X 0,Y 480.372,Z 457.882,A -85,B 0,C 180,E1 -7084.878,E2 -7084.878} C_VEL
LIN {X 0,Y 479.565,Z 462.435,A -85,B 0,C 180,E1 -7085.32,E2 -7085.32} C_VEL
LIN {X 0,Y 479.316,Z 472.55,A -85,B 0,C 180,E1 -7086.322,E2 -7086.322} C_VEL
LIN {X 0,Y 482.522,Z 492.251,A -85,B 0,C 180,E1 -7086.813,E2 -7086.813} C_VEL
LIN {X 0,Y 480.811,Z 640.401,A -85,B 0,C 180,E1 -7089.095,E2 -7089.095} C_VEL
LIN {X 0,Y 480.411,Z 656.314,A -85,B 0,C 180,E1 -7089.508,E2 -7089.508} C_VEL
LIN {X 0,Y 479.854,Z 670.237,A -85,B 0,C 180,E1 -7090.029,E2 -7090.029} C_VEL
LIN {X 0,Y 479.144,Z 684.518,A -85,B 0,C 180,E1 -7090.731,E2 -7090.731} C_VEL
LIN {X 0,Y 478.399,Z 698.258,A -85,B 0,C 180,E1 -7091.59,E2 -7091.59} C_VEL
LIN {X 0,Y 477.635,Z 710.885,A -85,B 0,C 180,E1 -7092.556,E2 -7092.556} C_VEL
LIN {X 0,Y 476.862,Z 723.636,A -85,B 0,C 180,E1 -7093.74,E2 -7093.74} C_VEL
LIN {X 0,Y 476.065,Z 735.197,A -85,B 0,C 180,E1 -7095.03,E2 -7095.03} C_VEL
LIN {X 0,Y 475.422,Z 744.943,A -85,B 0,C 180,E1 -7096.32,E2 -7096.32} C_VEL
LIN {X 0,Y 474.955,Z 754.014,A -85,B 0,C 180,E1 -7097.746,E2 -7097.746} C_VEL
LIN {X 0,Y 474.505,Z 762.423,A -85,B 0,C 180,E1 -7099.332,E2 -7099.332} C_VEL
LIN {X 0,Y 474.109,Z 769.832,A -85,B 0,C 180,E1 -7101.047,E2 -7101.047} C_VEL
LIN {X 0,Y 473.908,Z 775.717,A -85,B 0,C 180,E1 -7102.76,E2 -7102.76} C_VEL
LIN {X 0,Y 473.82,Z 779.189,A -85,B 0,C 180,E1 -7104.042,E2 -7104.042} C_VEL
LIN {X 0,Y 473.705,Z 782.728,A -85,B 0,C 180,E1 -7105.747,E2 -7105.747} C_VEL
LIN {X 0,Y 473.718,Z 785.069,A -85,B 0,C 180,E1 -7107.45,E2 -7107.45} C_VEL
LIN {X 0,Y 473.685,Z 786.264,A -85,B 0,C 180,E1 -7109.151,E2 -7109.151} C_VEL
LIN {X 0,Y 473.686,Z 786.281,A -85,B 0,C 180,E1 -7110.851,E2 -7110.851} C_VEL
LIN {X 0,Y 473.719,Z 785.155,A -85,B 0,C 180,E1 -7112.552,E2 -7112.552} C_VEL
LIN {X 0,Y 473.705,Z 782.879,A -85,B 0,C 180,E1 -7114.255,E2 -7114.255} C_VEL
LIN {X 0,Y 473.816,Z 779.402,A -85,B 0,C 180,E1 -7115.961,E2 -7115.961} C_VEL
LIN {X 0,Y 473.951,Z 774.643,A -85,B 0,C 180,E1 -7117.671,E2 -7117.671} C_VEL
LIN {X 0,Y 474.183,Z 768.481,A -85,B 0,C 180,E1 -7119.384,E2 -7119.384} C_VEL
LIN {X 0,Y 474.612,Z 760.73,A -85,B 0,C 180,E1 -7121.1,E2 -7121.1} C_VEL
LIN {X 0,Y 475.002,Z 752.474,A -85,B 0,C 180,E1 -7122.605,E2 -7122.605} C_VEL
LIN {X 0,Y 475.627,Z 742.508,A -85,B 0,C 180,E1 -7124.113,E2 -7124.113} C_VEL
LIN {X 0,Y 476.229,Z 732.348,A -85,B 0,C 180,E1 -7125.406,E2 -7125.406} C_VEL
LIN {X 0,Y 476.983,Z 720.952,A -85,B 0,C 180,E1 -7126.625,E2 -7126.625} C_VEL
LIN {X 0,Y 477.812,Z 708.046,A -85,B 0,C 180,E1 -7127.772,E2 -7127.772} C_VEL
LIN {X 0,Y 478.615,Z 694.826,A -85,B 0,C 180,E1 -7128.737,E2 -7128.737} C_VEL
LIN {X 0,Y 479.349,Z 681.223,A -85,B 0,C 180,E1 -7129.541,E2 -7129.541} C_VEL
LIN {X 0,Y 480.008,Z 666.319,A -85,B 0,C 180,E1 -7130.229,E2 -7130.229} C_VEL
LIN {X 0,Y 480.598,Z 651.01,A -85,B 0,C 180,E1 -7130.743,E2 -7130.743} C_VEL
LIN {X 0,Y 480.926,Z 635.279,A -85,B 0,C 180,E1 -7131.092,E2 -7131.092} C_VEL
LIN {X 0,Y 482.479,Z 491.439,A -85,B 0,C 180,E1 -7133.293,E2 -7133.293} C_VEL
LIN {X 0,Y 479.29,Z 472.305,A -85,B 0,C 180,E1 -7133.782,E2 -7133.782} C_VEL
LIN {X 0,Y 479.887,Z 452.379,A -85,B 0,C 180,E1 -7135.83,E2 -7135.83} C_VEL
LIN {X 0,Y 481.084,Z 424.672,A -85,B 0,C 180,E1 -7138.823,E2 -7138.823} C_VEL
LIN {X 0,Y 482.226,Z 399.029,A -85,B 0,C 180,E1 -7141.647,E2 -7141.647} C_VEL
LIN {X 0,Y 479.32,Z 387.781,A -85,B 0,C 180,E1 -7143.109,E2 -7143.109} C_VEL
LIN {X 0,Y 474.576,Z 372.176,A -85,B 0,C 180,E1 -7145.237,E2 -7145.237} C_VEL
LIN {X 0,Y 474.583,Z 371.991,A -85,B 0,C 180,E1 -7148.461,E2 -7148.461} C_VEL
LIN {X 0,Y 474.583,Z 371.983,A -85,B 0,C 180,E1 -7151.791,E2 -7151.791} C_VEL
LIN {X 0,Y 474.613,Z 371.988,A -85,B 0,C 180,E1 -7154.702,E2 -7154.702} C_VEL
LIN {X 0,Y 474.584,Z 371.991,A -85,B 0,C 180,E1 -7158.211,E2 -7158.211} C_VEL
LIN {X 0,Y 474.587,Z 371.994,A -85,B 0,C 180,E1 -7161.54,E2 -7161.54} C_VEL
LIN {X 0,Y 474.613,Z 371.977,A -85,B 0,C 180,E1 -7164.725,E2 -7164.725} C_VEL
LIN {X 0,Y 474.614,Z 371.988,A -85,B 0,C 180,E1 -7167.786,E2 -7167.786} C_VEL
LIN {X 0,Y 474.597,Z 371.994,A -85,B 0,C 180,E1 -7170.892,E2 -7170.892} C_VEL
LIN {X 0,Y 474.575,Z 371.995,A -85,B 0,C 180,E1 -7173.623,E2 -7173.623} C_VEL
LIN {X 0,Y 474.638,Z 371.988,A -85,B 0,C 180,E1 -7176.642,E2 -7176.642} C_VEL
LIN {X 0,Y 474.64,Z 372.155,A -85,B 0,C 180,E1 -7177.873,E2 -7177.873} C_VEL
LIN {X 0,Y 476.711,Z 381.803,A -85,B 0,C 180,E1 -7179.722,E2 -7179.722} C_VEL
LIN {X 0,Y 479.069,Z 390.159,A -85,B 0,C 180,E1 -7179.995,E2 -7179.995} C_VEL
LIN {X 0,Y 480.339,Z 396.61,A -85,B 0,C 180,E1 -7180.166,E2 -7180.166} C_VEL
LIN {X 0,Y 478.705,Z 521.115,A -85,B 0,C 180,E1 -7182.289,E2 -7182.289} C_VEL
LIN {X 0,Y 478.53,Z 536.001,A -85,B 0,C 180,E1 -7182.721,E2 -7182.721} C_VEL
LIN {X 0,Y 478.215,Z 549.82,A -85,B 0,C 180,E1 -7183.292,E2 -7183.292} C_VEL
LIN {X 0,Y 477.833,Z 562.746,A -85,B 0,C 180,E1 -7183.992,E2 -7183.992} C_VEL
LIN {X 0,Y 477.35,Z 573.92,A -85,B 0,C 180,E1 -7184.741,E2 -7184.741} C_VEL
LIN {X 0,Y 476.923,Z 585.696,A -85,B 0,C 180,E1 -7185.71,E2 -7185.71} C_VEL
LIN {X 0,Y 476.401,Z 596.851,A -85,B 0,C 180,E1 -7186.821,E2 -7186.821} C_VEL
LIN {X 0,Y 475.918,Z 607.199,A -85,B 0,C 180,E1 -7188.068,E2 -7188.068} C_VEL
LIN {X 0,Y 475.524,Z 616.012,A -85,B 0,C 180,E1 -7189.354,E2 -7189.354} C_VEL
LIN {X 0,Y 475.155,Z 624.445,A -85,B 0,C 180,E1 -7190.851,E2 -7190.851} C_VEL
LIN {X 0,Y 474.903,Z 631.2,A -85,B 0,C 180,E1 -7192.346,E2 -7192.346} C_VEL
LIN {X 0,Y 474.77,Z 635.882,A -85,B 0,C 180,E1 -7193.626,E2 -7193.626} C_VEL
LIN {X 0,Y 474.515,Z 639.626,A -85,B 0,C 180,E1 -7194.902,E2 -7194.902} C_VEL
LIN {X 0,Y 474.389,Z 643.319,A -85,B 0,C 180,E1 -7196.603,E2 -7196.603} C_VEL
LIN {X 0,Y 474.457,Z 644.615,A -85,B 0,C 180,E1 -7197.453,E2 -7197.453} C_VEL
LIN {X 0,Y 474.411,Z 646.214,A -85,B 0,C 180,E1 -7199.151,E2 -7199.151} C_VEL
LIN {X 0,Y 474.413,Z 646.458,A -85,B 0,C 180,E1 -7200.849,E2 -7200.849} C_VEL
LIN {X 0,Y 474.477,Z 645.334,A -85,B 0,C 180,E1 -7202.547,E2 -7202.547} C_VEL
LIN {X 0,Y 474.568,Z 642.841,A -85,B 0,C 180,E1 -7204.246,E2 -7204.246} C_VEL
LIN {X 0,Y 474.859,Z 638.881,A -85,B 0,C 180,E1 -7205.947,E2 -7205.947} C_VEL
LIN {X 0,Y 475.041,Z 634.891,A -85,B 0,C 180,E1 -7207.23,E2 -7207.23} C_VEL
LIN {X 0,Y 475.269,Z 629.957,A -85,B 0,C 180,E1 -7208.504,E2 -7208.504} C_VEL
LIN {X 0,Y 475.667,Z 622.753,A -85,B 0,C 180,E1 -7209.997,E2 -7209.997} C_VEL
LIN {X 0,Y 476.055,Z 615.176,A -85,B 0,C 180,E1 -7211.28,E2 -7211.28} C_VEL
LIN {X 0,Y 476.544,Z 605.965,A -85,B 0,C 180,E1 -7212.564,E2 -7212.564} C_VEL
LIN {X 0,Y 477.118,Z 595.753,A -85,B 0,C 180,E1 -7213.74,E2 -7213.74} C_VEL
LIN {X 0,Y 477.538,Z 584.497,A -85,B 0,C 180,E1 -7214.816,E2 -7214.816} C_VEL
LIN {X 0,Y 477.959,Z 572.003,A -85,B 0,C 180,E1 -7215.785,E2 -7215.785} C_VEL
LIN {X 0,Y 478.457,Z 559.847,A -85,B 0,C 180,E1 -7216.535,E2 -7216.535} C_VEL
LIN {X 0,Y 478.757,Z 547.285,A -85,B 0,C 180,E1 -7217.15,E2 -7217.15} C_VEL
LIN {X 0,Y 479.036,Z 532.948,A -85,B 0,C 180,E1 -7217.671,E2 -7217.671} C_VEL
LIN {X 0,Y 479.201,Z 518.304,A -85,B 0,C 180,E1 -7218.021,E2 -7218.021} C_VEL
LIN {X 0,Y 480.975,Z 432.509,A -85,B 0,C 180,E1 -7219.659,E2 -7219.659} C_VEL
LIN {X 0,Y 481.834,Z 397.332,A -85,B 0,C 180,E1 -7220.373,E2 -7220.373} C_VEL
LIN {X 0,Y 479.64,Z 390.67,A -85,B 0,C 180,E1 -7220.655,E2 -7220.655} C_VEL
LIN {X 0,Y 478.973,Z 388.913,A -85,B 0,C 180,E1 -7220.796,E2 -7220.796} C_VEL
LIN {X 0,Y 476.715,Z 379.488,A -85,B 0,C 180,E1 -7222.997,E2 -7222.997} C_VEL
LIN {X 0,Y 474.698,Z 372.049,A -85,B 0,C 180,E1 -7224.899,E2 -7224.899} C_VEL
LIN {X 0,Y 474.686,Z 371.983,A -85,B 0,C 180,E1 -7227.334,E2 -7227.334} C_VEL
LIN {X 0,Y 474.61,Z 371.993,A -85,B 0,C 180,E1 -7230.23,E2 -7230.23} C_VEL
LIN {X 0,Y 474.648,Z 371.987,A -85,B 0,C 180,E1 -7233.22,E2 -7233.22} C_VEL
LIN {X 0,Y 474.588,Z 371.996,A -85,B 0,C 180,E1 -7236.323,E2 -7236.323} C_VEL
LIN {X 0,Y 474.63,Z 371.988,A -85,B 0,C 180,E1 -7239.547,E2 -7239.547} C_VEL
LIN {X 0,Y 474.604,Z 371.994,A -85,B 0,C 180,E1 -7242.233,E2 -7242.233} C_VEL
LIN {X 0,Y 474.62,Z 371.989,A -85,B 0,C 180,E1 -7245.297,E2 -7245.297} C_VEL
LIN {X 0,Y 474.6,Z 371.996,A -85,B 0,C 180,E1 -7248.211,E2 -7248.211} C_VEL
LIN {X 0,Y 474.621,Z 371.992,A -85,B 0,C 180,E1 -7250.451,E2 -7250.451} C_VEL
LIN {X 0,Y 474.573,Z 371.998,A -85,B 0,C 180,E1 -7253.674,E2 -7253.674} C_VEL
LIN {X 0,Y 474.67,Z 372.173,A -85,B 0,C 180,E1 -7255.343,E2 -7255.343} C_VEL
LIN {X 0,Y 477.807,Z 381.807,A -85,B 0,C 180,E1 -7256.972,E2 -7256.972} C_VEL
LIN {X 0,Y 481.131,Z 394.05,A -85,B 0,C 180,E1 -7258.769,E2 -7258.769} C_VEL
LIN {X 0,Y 481.833,Z 398.099,A -85,B 0,C 180,E1 -7259.301,E2 -7259.301} C_VEL
LIN {X 0,Y 479.985,Z 426.239,A -85,B 0,C 180,E1 -7262.414,E2 -7262.414} C_VEL
LIN {X 0,Y 478.51,Z 457.383,A -85,B 0,C 180,E1 -7265.716,E2 -7265.716} C_VEL
LIN {X 0,Y 478.245,Z 463.492,A -85,B 0,C 180,E1 -7266.321,E2 -7266.321} C_VEL
LIN {X 0,Y 480.355,Z 479.815,A -85,B 0,C 180,E1 -7266.731,E2 -7266.731} C_VEL
LIN {X 0,Y 481.756,Z 491.321,A -85,B 0,C 180,E1 -7266.985,E2 -7266.985} C_VEL
LIN {X 0,Y 480.195,Z 641.322,A -85,B 0,C 180,E1 -7269.295,E2 -7269.295} C_VEL
LIN {X 0,Y 479.788,Z 657.229,A -85,B 0,C 180,E1 -7269.723,E2 -7269.723} C_VEL
LIN {X 0,Y 479.265,Z 671.791,A -85,B 0,C 180,E1 -7270.288,E2 -7270.288} C_VEL
LIN {X 0,Y 478.562,Z 686.403,A -85,B 0,C 180,E1 -7271.038,E2 -7271.038} C_VEL
LIN {X 0,Y 477.871,Z 699.655,A -85,B 0,C 180,E1 -7271.898,E2 -7271.898} C_VEL
LIN {X 0,Y 477.085,Z 713.204,A -85,B 0,C 180,E1 -7272.984,E2 -7272.984} C_VEL
LIN {X 0,Y 476.321,Z 725.296,A -85,B 0,C 180,E1 -7274.158,E2 -7274.158} C_VEL
LIN {X 0,Y 475.68,Z 736.403,A -85,B 0,C 180,E1 -7275.452,E2 -7275.452} C_VEL
LIN {X 0,Y 475.053,Z 747.151,A -85,B 0,C 180,E1 -7276.96,E2 -7276.96} C_VEL
LIN {X 0,Y 474.644,Z 756.078,A -85,B 0,C 180,E1 -7278.468,E2 -7278.468} C_VEL
LIN {X 0,Y 474.223,Z 764.411,A -85,B 0,C 180,E1 -7280.186,E2 -7280.186} C_VEL
LIN {X 0,Y 474.037,Z 771.081,A -85,B 0,C 180,E1 -7281.902,E2 -7281.902} C_VEL
LIN {X 0,Y 473.923,Z 776,A -85,B 0,C 180,E1 -7283.498,E2 -7283.498} C_VEL
LIN {X 0,Y 473.84,Z 779.292,A -85,B 0,C 180,E1 -7284.893,E2 -7284.893} C_VEL
LIN {X 0,Y 473.839,Z 782.229,A -85,B 0,C 180,E1 -7286.597,E2 -7286.597} C_VEL
LIN {X 0,Y 473.771,Z 783.979,A -85,B 0,C 180,E1 -7288.299,E2 -7288.299} C_VEL
LIN {X 0,Y 473.732,Z 784.575,A -85,B 0,C 180,E1 -7289.999,E2 -7289.999} C_VEL
LIN {X 0,Y 473.77,Z 783.978,A -85,B 0,C 180,E1 -7291.699,E2 -7291.699} C_VEL
LIN {X 0,Y 473.858,Z 782.227,A -85,B 0,C 180,E1 -7293.4,E2 -7293.4} C_VEL
LIN {X 0,Y 473.832,Z 779.295,A -85,B 0,C 180,E1 -7295.104,E2 -7295.104} C_VEL
LIN {X 0,Y 473.889,Z 775.11,A -85,B 0,C 180,E1 -7296.812,E2 -7296.812} C_VEL
LIN {X 0,Y 474.045,Z 769.557,A -85,B 0,C 180,E1 -7298.524,E2 -7298.524} C_VEL
LIN {X 0,Y 474.281,Z 762.484,A -85,B 0,C 180,E1 -7300.241,E2 -7300.241} C_VEL
LIN {X 0,Y 474.628,Z 754.901,A -85,B 0,C 180,E1 -7301.746,E2 -7301.746} C_VEL
LIN {X 0,Y 475.132,Z 745.753,A -85,B 0,C 180,E1 -7303.253,E2 -7303.253} C_VEL
LIN {X 0,Y 475.635,Z 736.422,A -85,B 0,C 180,E1 -7304.547,E2 -7304.547} C_VEL
LIN {X 0,Y 476.38,Z 724.301,A -85,B 0,C 180,E1 -7305.947,E2 -7305.947} C_VEL
LIN {X 0,Y 477.145,Z 711.897,A -85,B 0,C 180,E1 -7307.131,E2 -7307.131} C_VEL
LIN {X 0,Y 477.912,Z 698.128,A -85,B 0,C 180,E1 -7308.208,E2 -7308.208} C_VEL
LIN {X 0,Y 478.612,Z 684.531,A -85,B 0,C 180,E1 -7309.068,E2 -7309.068} C_VEL
LIN {X 0,Y 479.259,Z 670.442,A -85,B 0,C 180,E1 -7309.773,E2 -7309.773} C_VEL
LIN {X 0,Y 479.811,Z 655.766,A -85,B 0,C 180,E1 -7310.325,E2 -7310.325} C_VEL
LIN {X 0,Y 480.184,Z 641.432,A -85,B 0,C 180,E1 -7310.703,E2 -7310.703} C_VEL
LIN {X 0,Y 481.738,Z 490.201,A -85,B 0,C 180,E1 -7313.032,E2 -7313.032} C_VEL
LIN {X 0,Y 478.602,Z 467.355,A -85,B 0,C 180,E1 -7313.586,E2 -7313.586} C_VEL
LIN {X 0,Y 479.98,Z 438.187,A -85,B 0,C 180,E1 -7316.588,E2 -7316.588} C_VEL
LIN {X 0,Y 481.351,Z 410.296,A -85,B 0,C 180,E1 -7319.521,E2 -7319.521} C_VEL
LIN {X 0,Y 482.048,Z 398.246,A -85,B 0,C 180,E1 -7320.802,E2 -7320.802} C_VEL
LIN {X 0,Y 478.321,Z 384.598,A -85,B 0,C 180,E1 -7322.54,E2 -7322.54} C_VEL
LIN {X 0,Y 474.684,Z 372.175,A -85,B 0,C 180,E1 -7324.214,E2 -7324.214} C_VEL
LIN {X 0,Y 474.53,Z 372,A -85,B 0,C 180,E1 -7327.387,E2 -7327.387} C_VEL
LIN {X 0,Y 474.59,Z 371.993,A -85,B 0,C 180,E1 -7329.642,E2 -7329.642} C_VEL
LIN {X 0,Y 474.563,Z 371.995,A -85,B 0,C 180,E1 -7332.938,E2 -7332.938} C_VEL
LIN {X 0,Y 474.585,Z 371.993,A -85,B 0,C 180,E1 -7335.892,E2 -7335.892} C_VEL
LIN {X 0,Y 474.577,Z 371.985,A -85,B 0,C 180,E1 -7339.338,E2 -7339.338} C_VEL
LIN {X 0,Y 474.576,Z 371.993,A -85,B 0,C 180,E1 -7341.706,E2 -7341.706} C_VEL
LIN {X 0,Y 474.596,Z 371.966,A -85,B 0,C 180,E1 -7344.723,E2 -7344.723} C_VEL
LIN {X 0,Y 474.613,Z 371.985,A -85,B 0,C 180,E1 -7347.786,E2 -7347.786} C_VEL
LIN {X 0,Y 474.583,Z 371.988,A -85,B 0,C 180,E1 -7350.89,E2 -7350.89} C_VEL
LIN {X 0,Y 474.577,Z 371.991,A -85,B 0,C 180,E1 -7353.623,E2 -7353.623} C_VEL
LIN {X 0,Y 474.619,Z 371.991,A -85,B 0,C 180,E1 -7356.641,E2 -7356.641} C_VEL
LIN {X 0,Y 474.631,Z 371.98,A -85,B 0,C 180,E1 -7360.089,E2 -7360.089} C_VEL
LIN {X 0,Y 474.576,Z 371.994,A -85,B 0,C 180,E1 -7362.772,E2 -7362.772} C_VEL
LIN {X 0,Y 474.615,Z 371.978,A -85,B 0,C 180,E1 -7365.42,E2 -7365.42} C_VEL
LIN {X 0,Y 474.687,Z 371.98,A -85,B 0,C 180,E1 -7368.037,E2 -7368.037} C_VEL
LIN {X 0,Y 474.649,Z 371.977,A -85,B 0,C 180,E1 -7371.485,E2 -7371.485} C_VEL
LIN {X 0,Y 474.711,Z 371.976,A -85,B 0,C 180,E1 -7374.052,E2 -7374.052} C_VEL
LIN {X 0,Y 474.863,Z 371.954,A -85,B 0,C 180,E1 -7377.455,E2 -7377.455} C_VEL
LIN {X 0,Y 474.8,Z 371.957,A -85,B 0,C 180,E1 -7380.848,E2 -7380.848} C_VEL
LIN {X 0,Y 474.86,Z 371.956,A -85,B 0,C 180,E1 -7382.545,E2 -7382.545} C_VEL
LIN {X 0,Y 474.74,Z 371.968,A -85,B 0,C 180,E1 -7385.948,E2 -7385.948} C_VEL
LIN {X 0,Y 474.685,Z 371.98,A -85,B 0,C 180,E1 -7388.514,E2 -7388.514} C_VEL
LIN {X 0,Y 474.687,Z 371.968,A -85,B 0,C 180,E1 -7391.963,E2 -7391.963} C_VEL
LIN {X 0,Y 474.664,Z 371.976,A -85,B 0,C 180,E1 -7395.768,E2 -7395.768} C_VEL
LIN {X 0,Y 474.646,Z 371.985,A -85,B 0,C 180,E1 -7399.011,E2 -7399.011} C_VEL
LIN {X 0,Y 474.573,Z 371.986,A -85,B 0,C 180,E1 -7401.73,E2 -7401.73} C_VEL
LIN {X 0,Y 474.609,Z 371.991,A -85,B 0,C 180,E1 -7404.496,E2 -7404.496} C_VEL
LIN {X 0,Y 474.583,Z 371.992,A -85,B 0,C 180,E1 -7407.327,E2 -7407.327} C_VEL
LIN {X 0,Y 474.566,Z 371.992,A -85,B 0,C 180,E1 -7410.233,E2 -7410.233} C_VEL
LIN {X 0,Y 474.6,Z 371.992,A -85,B 0,C 180,E1 -7413.224,E2 -7413.224} C_VEL
LIN {X 0,Y 474.568,Z 371.988,A -85,B 0,C 180,E1 -7416.326,E2 -7416.326} C_VEL
LIN {X 0,Y 474.588,Z 371.991,A -85,B 0,C 180,E1 -7419.645,E2 -7419.645} C_VEL
LIN {X 0,Y 474.563,Z 371.984,A -85,B 0,C 180,E1 -7422.231,E2 -7422.231} C_VEL
LIN {X 0,Y 474.601,Z 371.989,A -85,B 0,C 180,E1 -7425.3,E2 -7425.3} C_VEL
LIN {X 0,Y 474.581,Z 371.994,A -85,B 0,C 180,E1 -7428.213,E2 -7428.213} C_VEL
LIN {X 0,Y 474.608,Z 371.982,A -85,B 0,C 180,E1 -7430.453,E2 -7430.453} C_VEL
LIN {X 0,Y 474.562,Z 371.993,A -85,B 0,C 180,E1 -7433.676,E2 -7433.676} C_VEL
LIN {X 0,Y 474.646,Z 372.204,A -85,B 0,C 180,E1 -7434.874,E2 -7434.874} C_VEL
LIN {X 0,Y 479.286,Z 387.671,A -85,B 0,C 180,E1 -7436.979,E2 -7436.979} C_VEL
LIN {X 0,Y 482.16,Z 398.187,A -85,B 0,C 180,E1 -7438.351,E2 -7438.351} C_VEL
LIN {X 0,Y 481.334,Z 417.478,A -85,B 0,C 180,E1 -7440.478,E2 -7440.478} C_VEL
LIN {X 0,Y 480.289,Z 442.445,A -85,B 0,C 180,E1 -7443.203,E2 -7443.203} C_VEL
LIN {X 0,Y 479.565,Z 462.435,A -85,B 0,C 180,E1 -7445.32,E2 -7445.32} C_VEL
LIN {X 0,Y 478.861,Z 465.678,A -85,B 0,C 180,E1 -7445.596,E2 -7445.596} C_VEL
LIN {X 0,Y 476.333,Z 471.492,A -85,B 0,C 180,E1 -7445.906,E2 -7445.906} C_VEL
LIN {X 0,Y 474.494,Z 476.454,A -85,B 0,C 180,E1 -7446.072,E2 -7446.072} C_VEL
LIN {X 0,Y 474.023,Z 480.355,A -85,B 0,C 180,E1 -7446.176,E2 -7446.176} C_VEL
LIN {X 0,Y 474.158,Z 481.66,A -85,B 0,C 180,E1 -7446.21,E2 -7446.21} C_VEL
LIN {X 0,Y 475.994,Z 493.084,A -85,B 0,C 180,E1 -7446.491,E2 -7446.491} C_VEL
LIN {X 0,Y 474.179,Z 640.297,A -85,B 0,C 180,E1 -7448.788,E2 -7448.788} C_VEL
LIN {X 0,Y 473.752,Z 656.028,A -85,B 0,C 180,E1 -7449.2,E2 -7449.2} C_VEL
LIN {X 0,Y 473.17,Z 670.496,A -85,B 0,C 180,E1 -7449.748,E2 -7449.748} C_VEL
LIN {X 0,Y 472.438,Z 684.481,A -85,B 0,C 180,E1 -7450.447,E2 -7450.447} C_VEL
LIN {X 0,Y 471.616,Z 698.227,A -85,B 0,C 180,E1 -7451.315,E2 -7451.315} C_VEL
LIN {X 0,Y 470.74,Z 712.12,A -85,B 0,C 180,E1 -7452.404,E2 -7452.404} C_VEL
LIN {X 0,Y 469.923,Z 724.659,A -85,B 0,C 180,E1 -7453.605,E2 -7453.605} C_VEL
LIN {X 0,Y 469.135,Z 735.176,A -85,B 0,C 180,E1 -7454.803,E2 -7454.803} C_VEL
LIN {X 0,Y 468.356,Z 746.384,A -85,B 0,C 180,E1 -7456.331,E2 -7456.331} C_VEL
LIN {X 0,Y 467.837,Z 755.671,A -85,B 0,C 180,E1 -7457.861,E2 -7457.861} C_VEL
LIN {X 0,Y 467.495,Z 762.406,A -85,B 0,C 180,E1 -7459.17,E2 -7459.17} C_VEL
LIN {X 0,Y 467.068,Z 769.816,A -85,B 0,C 180,E1 -7460.911,E2 -7460.911} C_VEL
LIN {X 0,Y 466.826,Z 775.702,A -85,B 0,C 180,E1 -7462.649,E2 -7462.649} C_VEL
LIN {X 0,Y 466.731,Z 779.174,A -85,B 0,C 180,E1 -7463.951,E2 -7463.951} C_VEL
LIN {X 0,Y 466.618,Z 782.714,A -85,B 0,C 180,E1 -7465.682,E2 -7465.682} C_VEL
LIN {X 0,Y 466.639,Z 785.056,A -85,B 0,C 180,E1 -7467.412,E2 -7467.412} C_VEL
LIN {X 0,Y 466.586,Z 786.25,A -85,B 0,C 180,E1 -7469.138,E2 -7469.138} C_VEL
LIN {X 0,Y 466.587,Z 786.267,A -85,B 0,C 180,E1 -7470.864,E2 -7470.864} C_VEL
LIN {X 0,Y 466.64,Z 785.14,A -85,B 0,C 180,E1 -7472.591,E2 -7472.591} C_VEL
LIN {X 0,Y 466.618,Z 782.863,A -85,B 0,C 180,E1 -7474.32,E2 -7474.32} C_VEL
LIN {X 0,Y 466.736,Z 779.385,A -85,B 0,C 180,E1 -7476.052,E2 -7476.052} C_VEL
LIN {X 0,Y 466.887,Z 774.624,A -85,B 0,C 180,E1 -7477.787,E2 -7477.787} C_VEL
LIN {X 0,Y 467.126,Z 768.46,A -85,B 0,C 180,E1 -7479.527,E2 -7479.527} C_VEL
LIN {X 0,Y 467.6,Z 760.706,A -85,B 0,C 180,E1 -7481.269,E2 -7481.269} C_VEL
LIN {X 0,Y 468.003,Z 752.314,A -85,B 0,C 180,E1 -7482.819,E2 -7482.819} C_VEL
LIN {X 0,Y 468.675,Z 742.479,A -85,B 0,C 180,E1 -7484.326,E2 -7484.326} C_VEL
LIN {X 0,Y 469.325,Z 732.317,A -85,B 0,C 180,E1 -7485.638,E2 -7485.638} C_VEL
LIN {X 0,Y 470.22,Z 720.105,A -85,B 0,C 180,E1 -7486.95,E2 -7486.95} C_VEL
LIN {X 0,Y 471.009,Z 708.005,A -85,B 0,C 180,E1 -7488.037,E2 -7488.037} C_VEL
LIN {X 0,Y 471.835,Z 694.777,A -85,B 0,C 180,E1 -7489.017,E2 -7489.017} C_VEL
LIN {X 0,Y 472.646,Z 681.166,A -85,B 0,C 180,E1 -7489.83,E2 -7489.83} C_VEL
LIN {X 0,Y 473.361,Z 665.972,A -85,B 0,C 180,E1 -7490.536,E2 -7490.536} C_VEL
LIN {X 0,Y 473.955,Z 650.894,A -85,B 0,C 180,E1 -7491.048,E2 -7491.048} C_VEL
LIN {X 0,Y 474.331,Z 635.092,A -85,B 0,C 180,E1 -7491.4,E2 -7491.4} C_VEL
LIN {X 0,Y 475.943,Z 492.349,A -85,B 0,C 180,E1 -7493.615,E2 -7493.615} C_VEL
LIN {X 0,Y 472.594,Z 472.187,A -85,B 0,C 180,E1 -7494.14,E2 -7494.14} C_VEL
LIN {X 0,Y 473.337,Z 449.958,A -85,B 0,C 180,E1 -7496.452,E2 -7496.452} C_VEL
LIN {X 0,Y 474.523,Z 423.201,A -85,B 0,C 180,E1 -7499.381,E2 -7499.381} C_VEL
LIN {X 0,Y 475.543,Z 400.599,A -85,B 0,C 180,E1 -7501.895,E2 -7501.895} C_VEL
LIN {X 0,Y 471.387,Z 385.519,A -85,B 0,C 180,E1 -7503.905,E2 -7503.905} C_VEL
LIN {X 0,Y 467.54,Z 373.134,A -85,B 0,C 180,E1 -7505.624,E2 -7505.624} C_VEL
LIN {X 0,Y 467.511,Z 372.873,A -85,B 0,C 180,E1 -7505.894,E2 -7505.894} C_VEL
LIN {X 0,Y 467.529,Z 372.866,A -85,B 0,C 180,E1 -7509.151,E2 -7509.151} C_VEL
LIN {X 0,Y 467.553,Z 372.862,A -85,B 0,C 180,E1 -7511.407,E2 -7511.407} C_VEL
LIN {X 0,Y 467.557,Z 372.861,A -85,B 0,C 180,E1 -7515.051,E2 -7515.051} C_VEL
LIN {X 0,Y 467.554,Z 372.867,A -85,B 0,C 180,E1 -7518.728,E2 -7518.728} C_VEL
LIN {X 0,Y 467.541,Z 372.869,A -85,B 0,C 180,E1 -7521.953,E2 -7521.953} C_VEL
LIN {X 0,Y 467.548,Z 372.853,A -85,B 0,C 180,E1 -7525.166,E2 -7525.166} C_VEL
LIN {X 0,Y 467.549,Z 372.868,A -85,B 0,C 180,E1 -7528.257,E2 -7528.257} C_VEL
LIN {X 0,Y 467.543,Z 372.873,A -85,B 0,C 180,E1 -7531.248,E2 -7531.248} C_VEL
LIN {X 0,Y 467.565,Z 372.868,A -85,B 0,C 180,E1 -7534.406,E2 -7534.406} C_VEL
LIN {X 0,Y 467.6,Z 372.978,A -85,B 0,C 180,E1 -7537.61,E2 -7537.61} C_VEL
LIN {X 0,Y 469.644,Z 382.297,A -85,B 0,C 180,E1 -7539.412,E2 -7539.412} C_VEL
LIN {X 0,Y 472.325,Z 391.035,A -85,B 0,C 180,E1 -7539.722,E2 -7539.722} C_VEL
LIN {X 0,Y 473.649,Z 397.126,A -85,B 0,C 180,E1 -7539.891,E2 -7539.891} C_VEL
LIN {X 0,Y 471.871,Z 522.46,A -85,B 0,C 180,E1 -7542.082,E2 -7542.082} C_VEL
LIN {X 0,Y 471.696,Z 537.136,A -85,B 0,C 180,E1 -7542.521,E2 -7542.521} C_VEL
LIN {X 0,Y 471.372,Z 550.805,A -85,B 0,C 180,E1 -7543.098,E2 -7543.098} C_VEL
LIN {X 0,Y 470.914,Z 564.587,A -85,B 0,C 180,E1 -7543.861,E2 -7543.861} C_VEL
LIN {X 0,Y 470.437,Z 577.026,A -85,B 0,C 180,E1 -7544.734,E2 -7544.734} C_VEL
LIN {X 0,Y 469.933,Z 588.442,A -85,B 0,C 180,E1 -7545.714,E2 -7545.714} C_VEL
LIN {X 0,Y 469.411,Z 599.771,A -85,B 0,C 180,E1 -7546.895,E2 -7546.895} C_VEL
LIN {X 0,Y 468.937,Z 609.392,A -85,B 0,C 180,E1 -7548.108,E2 -7548.108} C_VEL
LIN {X 0,Y 468.493,Z 618.014,A -85,B 0,C 180,E1 -7549.411,E2 -7549.411} C_VEL
LIN {X 0,Y 468.17,Z 626.234,A -85,B 0,C 180,E1 -7550.931,E2 -7550.931} C_VEL
LIN {X 0,Y 467.858,Z 633.05,A -85,B 0,C 180,E1 -7552.497,E2 -7552.497} C_VEL
LIN {X 0,Y 467.618,Z 638.101,A -85,B 0,C 180,E1 -7553.961,E2 -7553.961} C_VEL
LIN {X 0,Y 467.41,Z 642.588,A -85,B 0,C 180,E1 -7555.688,E2 -7555.688} C_VEL
LIN {X 0,Y 467.442,Z 645.593,A -85,B 0,C 180,E1 -7557.415,E2 -7557.415} C_VEL
LIN {X 0,Y 467.395,Z 647.237,A -85,B 0,C 180,E1 -7559.138,E2 -7559.138} C_VEL
LIN {X 0,Y 467.399,Z 647.521,A -85,B 0,C 180,E1 -7560.861,E2 -7560.861} C_VEL
LIN {X 0,Y 467.494,Z 646.421,A -85,B 0,C 180,E1 -7562.585,E2 -7562.585} C_VEL
LIN {X 0,Y 467.571,Z 643.949,A -85,B 0,C 180,E1 -7564.31,E2 -7564.31} C_VEL
LIN {X 0,Y 467.883,Z 639.998,A -85,B 0,C 180,E1 -7566.035,E2 -7566.035} C_VEL
LIN {X 0,Y 468.1,Z 635.904,A -85,B 0,C 180,E1 -7567.367,E2 -7567.367} C_VEL
LIN {X 0,Y 468.331,Z 631.074,A -85,B 0,C 180,E1 -7568.631,E2 -7568.631} C_VEL
LIN {X 0,Y 468.763,Z 623.879,A -85,B 0,C 180,E1 -7570.146,E2 -7570.146} C_VEL
LIN {X 0,Y 469.192,Z 616.33,A -85,B 0,C 180,E1 -7571.447,E2 -7571.447} C_VEL
LIN {X 0,Y 469.735,Z 607.153,A -85,B 0,C 180,E1 -7572.749,E2 -7572.749} C_VEL
LIN {X 0,Y 470.334,Z 596.943,A -85,B 0,C 180,E1 -7573.942,E2 -7573.942} C_VEL
LIN {X 0,Y 470.783,Z 585.68,A -85,B 0,C 180,E1 -7575.033,E2 -7575.033} C_VEL
LIN {X 0,Y 471.226,Z 573.185,A -85,B 0,C 180,E1 -7576.016,E2 -7576.016} C_VEL
LIN {X 0,Y 471.823,Z 559.156,A -85,B 0,C 180,E1 -7576.885,E2 -7576.885} C_VEL
LIN {X 0,Y 472.206,Z 546.565,A -85,B 0,C 180,E1 -7577.489,E2 -7577.489} C_VEL
LIN {X 0,Y 472.416,Z 531.956,A -85,B 0,C 180,E1 -7578.005,E2 -7578.005} C_VEL
LIN {X 0,Y 472.568,Z 516.232,A -85,B 0,C 180,E1 -7578.367,E2 -7578.367} C_VEL
LIN {X 0,Y 474.567,Z 432.104,A -85,B 0,C 180,E1 -7580.028,E2 -7580.028} C_VEL
LIN {X 0,Y 475.458,Z 398.819,A -85,B 0,C 180,E1 -7580.731,E2 -7580.731} C_VEL
LIN {X 0,Y 473.606,Z 393.467,A -85,B 0,C 180,E1 -7580.977,E2 -7580.977} C_VEL
LIN {X 0,Y 472.171,Z 390.278,A -85,B 0,C 180,E1 -7581.187,E2 -7581.187} C_VEL
LIN {X 0,Y 469.533,Z 379.819,A -85,B 0,C 180,E1 -7583.708,E2 -7583.708} C_VEL
LIN {X 0,Y 467.639,Z 372.916,A -85,B 0,C 180,E1 -7585.564,E2 -7585.564} C_VEL
LIN {X 0,Y 467.625,Z 372.861,A -85,B 0,C 180,E1 -7587.769,E2 -7587.769} C_VEL
LIN {X 0,Y 467.573,Z 372.87,A -85,B 0,C 180,E1 -7591.044,E2 -7591.044} C_VEL
LIN {X 0,Y 467.593,Z 372.868,A -85,B 0,C 180,E1 -7594.242,E2 -7594.242} C_VEL
LIN {X 0,Y 467.547,Z 372.87,A -85,B 0,C 180,E1 -7597.185,E2 -7597.185} C_VEL
LIN {X 0,Y 467.575,Z 372.869,A -85,B 0,C 180,E1 -7600.265,E2 -7600.265} C_VEL
LIN {X 0,Y 467.552,Z 372.871,A -85,B 0,C 180,E1 -7603.745,E2 -7603.745} C_VEL
LIN {X 0,Y 467.55,Z 372.873,A -85,B 0,C 180,E1 -7606.254,E2 -7606.254} C_VEL
LIN {X 0,Y 467.56,Z 372.871,A -85,B 0,C 180,E1 -7609.732,E2 -7609.732} C_VEL
LIN {X 0,Y 467.518,Z 372.876,A -85,B 0,C 180,E1 -7612.818,E2 -7612.818} C_VEL
LIN {X 0,Y 467.595,Z 373.055,A -85,B 0,C 180,E1 -7614.742,E2 -7614.742} C_VEL
LIN {X 0,Y 470.12,Z 380.508,A -85,B 0,C 180,E1 -7616.099,E2 -7616.099} C_VEL
LIN {X 0,Y 473.482,Z 391.909,A -85,B 0,C 180,E1 -7617.913,E2 -7617.913} C_VEL
LIN {X 0,Y 475.279,Z 399.926,A -85,B 0,C 180,E1 -7619.054,E2 -7619.054} C_VEL
LIN {X 0,Y 473.369,Z 426.954,A -85,B 0,C 180,E1 -7622.116,E2 -7622.116} C_VEL
LIN {X 0,Y 471.678,Z 458.16,A -85,B 0,C 180,E1 -7625.494,E2 -7625.494} C_VEL
LIN {X 0,Y 471.515,Z 462.415,A -85,B 0,C 180,E1 -7625.923,E2 -7625.923} C_VEL
LIN {X 0,Y 473.69,Z 479.002,A -85,B 0,C 180,E1 -7626.368,E2 -7626.368} C_VEL
LIN {X 0,Y 475.235,Z 491.476,A -85,B 0,C 180,E1 -7626.651,E2 -7626.651} C_VEL
LIN {X 0,Y 473.636,Z 638.53,A -85,B 0,C 180,E1 -7628.938,E2 -7628.938} C_VEL
LIN {X 0,Y 473.247,Z 653.269,A -85,B 0,C 180,E1 -7629.299,E2 -7629.299} C_VEL
LIN {X 0,Y 472.728,Z 667.689,A -85,B 0,C 180,E1 -7629.819,E2 -7629.819} C_VEL
LIN {X 0,Y 472.02,Z 682.567,A -85,B 0,C 180,E1 -7630.539,E2 -7630.539} C_VEL
LIN {X 0,Y 471.283,Z 696.562,A -85,B 0,C 180,E1 -7631.411,E2 -7631.411} C_VEL
LIN {X 0,Y 470.493,Z 709.32,A -85,B 0,C 180,E1 -7632.392,E2 -7632.392} C_VEL
LIN {X 0,Y 469.679,Z 722.168,A -85,B 0,C 180,E1 -7633.593,E2 -7633.593} C_VEL
LIN {X 0,Y 468.959,Z 732.897,A -85,B 0,C 180,E1 -7634.795,E2 -7634.795} C_VEL
LIN {X 0,Y 468.376,Z 742.796,A -85,B 0,C 180,E1 -7636.108,E2 -7636.108} C_VEL
LIN {X 0,Y 467.767,Z 752.139,A -85,B 0,C 180,E1 -7637.579,E2 -7637.579} C_VEL
LIN {X 0,Y 467.429,Z 760.488,A -85,B 0,C 180,E1 -7639.166,E2 -7639.166} C_VEL
LIN {X 0,Y 467.065,Z 767.958,A -85,B 0,C 180,E1 -7640.908,E2 -7640.908} C_VEL
LIN {X 0,Y 466.846,Z 773.876,A -85,B 0,C 180,E1 -7642.647,E2 -7642.647} C_VEL
LIN {X 0,Y 466.798,Z 777.373,A -85,B 0,C 180,E1 -7643.949,E2 -7643.949} C_VEL
LIN {X 0,Y 466.715,Z 780.928,A -85,B 0,C 180,E1 -7645.681,E2 -7645.681} C_VEL
LIN {X 0,Y 466.722,Z 783.263,A -85,B 0,C 180,E1 -7647.409,E2 -7647.409} C_VEL
LIN {X 0,Y 466.672,Z 784.436,A -85,B 0,C 180,E1 -7649.136,E2 -7649.136} C_VEL
LIN {X 0,Y 466.672,Z 784.436,A -85,B 0,C 180,E1 -7650.862,E2 -7650.862} C_VEL
LIN {X 0,Y 466.721,Z 783.261,A -85,B 0,C 180,E1 -7652.588,E2 -7652.588} C_VEL
LIN {X 0,Y 466.695,Z 780.928,A -85,B 0,C 180,E1 -7654.317,E2 -7654.317} C_VEL
LIN {X 0,Y 466.77,Z 777.381,A -85,B 0,C 180,E1 -7656.049,E2 -7656.049} C_VEL
LIN {X 0,Y 466.903,Z 772.53,A -85,B 0,C 180,E1 -7657.784,E2 -7657.784} C_VEL
LIN {X 0,Y 467.118,Z 766.241,A -85,B 0,C 180,E1 -7659.525,E2 -7659.525} C_VEL
LIN {X 0,Y 467.527,Z 758.334,A -85,B 0,C 180,E1 -7661.268,E2 -7661.268} C_VEL
LIN {X 0,Y 467.918,Z 749.755,A -85,B 0,C 180,E1 -7662.82,E2 -7662.82} C_VEL
LIN {X 0,Y 468.504,Z 739.693,A -85,B 0,C 180,E1 -7664.329,E2 -7664.329} C_VEL
LIN {X 0,Y 469.14,Z 729.24,A -85,B 0,C 180,E1 -7665.642,E2 -7665.642} C_VEL
LIN {X 0,Y 469.924,Z 717.947,A -85,B 0,C 180,E1 -7666.832,E2 -7666.832} C_VEL
LIN {X 0,Y 470.724,Z 705.413,A -85,B 0,C 180,E1 -7667.933,E2 -7667.933} C_VEL
LIN {X 0,Y 471.477,Z 691.748,A -85,B 0,C 180,E1 -7668.916,E2 -7668.916} C_VEL
LIN {X 0,Y 472.266,Z 677.51,A -85,B 0,C 180,E1 -7669.73,E2 -7669.73} C_VEL
LIN {X 0,Y 472.897,Z 662.404,A -85,B 0,C 180,E1 -7670.394,E2 -7670.394} C_VEL
LIN {X 0,Y 473.381,Z 647.21,A -85,B 0,C 180,E1 -7670.872,E2 -7670.872} C_VEL
LIN {X 0,Y 473.712,Z 630.657,A -85,B 0,C 180,E1 -7671.198,E2 -7671.198} C_VEL
LIN {X 0,Y 475.215,Z 491.796,A -85,B 0,C 180,E1 -7673.344,E2 -7673.344} C_VEL
LIN {X 0,Y 471.87,Z 466.685,A -85,B 0,C 180,E1 -7673.943,E2 -7673.943} C_VEL
LIN {X 0,Y 473.209,Z 438.644,A -85,B 0,C 180,E1 -7676.858,E2 -7676.858} C_VEL
LIN {X 0,Y 474.778,Z 409.486,A -85,B 0,C 180,E1 -7679.971,E2 -7679.971} C_VEL
LIN {X 0,Y 475.355,Z 400.271,A -85,B 0,C 180,E1 -7680.961,E2 -7680.961} C_VEL
LIN {X 0,Y 471.439,Z 385.953,A -85,B 0,C 180,E1 -7682.817,E2 -7682.817} C_VEL
LIN {X 0,Y 467.612,Z 373.023,A -85,B 0,C 180,E1 -7684.603,E2 -7684.603} C_VEL
LIN {X 0,Y 467.53,Z 372.875,A -85,B 0,C 180,E1 -7688.046,E2 -7688.046} C_VEL
LIN {X 0,Y 467.551,Z 372.868,A -85,B 0,C 180,E1 -7691.273,E2 -7691.273} C_VEL
LIN {X 0,Y 467.551,Z 372.868,A -85,B 0,C 180,E1 -7694.947,E2 -7694.947} C_VEL
LIN {X 0,Y 467.547,Z 372.854,A -85,B 0,C 180,E1 -7698.725,E2 -7698.725} C_VEL
LIN {X 0,Y 467.526,Z 372.873,A -85,B 0,C 180,E1 -7701.952,E2 -7701.952} C_VEL
LIN {X 0,Y 467.535,Z 372.845,A -85,B 0,C 180,E1 -7705.165,E2 -7705.165} C_VEL
LIN {X 0,Y 467.563,Z 372.869,A -85,B 0,C 180,E1 -7708.258,E2 -7708.258} C_VEL
LIN {X 0,Y 467.529,Z 372.865,A -85,B 0,C 180,E1 -7711.247,E2 -7711.247} C_VEL
LIN {X 0,Y 467.563,Z 372.864,A -85,B 0,C 180,E1 -7714.4,E2 -7714.4} C_VEL
LIN {X 0,Y 467.556,Z 372.867,A -85,B 0,C 180,E1 -7716.995,E2 -7716.995} C_VEL
LIN {X 0,Y 467.602,Z 372.855,A -85,B 0,C 180,E1 -7719.776,E2 -7719.776} C_VEL
LIN {X 0,Y 467.548,Z 372.874,A -85,B 0,C 180,E1 -7722.505,E2 -7722.505} C_VEL
LIN {X 0,Y 467.574,Z 372.856,A -85,B 0,C 180,E1 -7725.195,E2 -7725.195} C_VEL
LIN {X 0,Y 467.639,Z 372.856,A -85,B 0,C 180,E1 -7727.854,E2 -7727.854} C_VEL
LIN {X 0,Y 467.618,Z 372.853,A -85,B 0,C 180,E1 -7731.356,E2 -7731.356} C_VEL
LIN {X 0,Y 467.676,Z 372.851,A -85,B 0,C 180,E1 -7733.962,E2 -7733.962} C_VEL
LIN {X 0,Y 467.804,Z 372.833,A -85,B 0,C 180,E1 -7737.417,E2 -7737.417} C_VEL
LIN {X 0,Y 467.83,Z 372.831,A -85,B 0,C 180,E1 -7740,E2 -7740} C_VEL
LIN {X 0,Y 467.801,Z 372.835,A -85,B 0,C 180,E1 -7742.583,E2 -7742.583} C_VEL
LIN {X 0,Y 467.705,Z 372.845,A -85,B 0,C 180,E1 -7746.038,E2 -7746.038} C_VEL
LIN {X 0,Y 467.643,Z 372.859,A -85,B 0,C 180,E1 -7748.644,E2 -7748.644} C_VEL
LIN {X 0,Y 467.639,Z 372.847,A -85,B 0,C 180,E1 -7752.146,E2 -7752.146} C_VEL
LIN {X 0,Y 467.633,Z 372.852,A -85,B 0,C 180,E1 -7755.885,E2 -7755.885} C_VEL
LIN {X 0,Y 467.606,Z 372.859,A -85,B 0,C 180,E1 -7759.309,E2 -7759.309} C_VEL
LIN {X 0,Y 467.516,Z 372.867,A -85,B 0,C 180,E1 -7762.075,E2 -7762.075} C_VEL
LIN {X 0,Y 467.539,Z 372.866,A -85,B 0,C 180,E1 -7764.891,E2 -7764.891} C_VEL
LIN {X 0,Y 467.529,Z 372.87,A -85,B 0,C 180,E1 -7767.775,E2 -7767.775} C_VEL
LIN {X 0,Y 467.523,Z 372.875,A -85,B 0,C 180,E1 -7771.039,E2 -7771.039} C_VEL
LIN {X 0,Y 467.563,Z 372.868,A -85,B 0,C 180,E1 -7774.241,E2 -7774.241} C_VEL
LIN {X 0,Y 467.509,Z 372.855,A -85,B 0,C 180,E1 -7777.183,E2 -7777.183} C_VEL
LIN {X 0,Y 467.544,Z 372.871,A -85,B 0,C 180,E1 -7780.268,E2 -7780.268} C_VEL
LIN {X 0,Y 467.521,Z 372.87,A -85,B 0,C 180,E1 -7783.749,E2 -7783.749} C_VEL
LIN {X 0,Y 467.521,Z 372.866,A -85,B 0,C 180,E1 -7786.254,E2 -7786.254} C_VEL
LIN {X 0,Y 467.55,Z 372.874,A -85,B 0,C 180,E1 -7788.727,E2 -7788.727} C_VEL
LIN {X 0,Y 467.531,Z 372.873,A -85,B 0,C 180,E1 -7791.955,E2 -7791.955} C_VEL
LIN {X 0,Y 467.59,Z 373.067,A -85,B 0,C 180,E1 -7794.458,E2 -7794.458} C_VEL
LIN {X 0,Y 472.257,Z 388.435,A -85,B 0,C 180,E1 -7796.592,E2 -7796.592} C_VEL
LIN {X 0,Y 475.548,Z 400.905,A -85,B 0,C 180,E1 -7798.233,E2 -7798.233} C_VEL
LIN {X 0,Y 474.302,Z 428.677,A -85,B 0,C 180,E1 -7801.326,E2 -7801.326} C_VEL
LIN {X 0,Y 472.946,Z 461.36,A -85,B 0,C 180,E1 -7804.852,E2 -7804.852} C_VEL
LIN {X 0,Y 472.617,Z 472.456,A -85,B 0,C 180,E1 -7805.966,E2 -7805.966} C_VEL
LIN {X 0,Y 474.158,Z 481.66,A -85,B 0,C 180,E1 -7806.21,E2 -7806.21} C_VEL
LIN {X 0,Y 474.374,Z 487.477,A -85,B 0,C 180,E1 -7806.316,E2 -7806.316} C_VEL
LIN {X 0,Y 473.442,Z 493.338,A -85,B 0,C 180,E1 -7806.362,E2 -7806.362} C_VEL
LIN {X 0,Y 470.38,Z 505.028,A -85,B 0,C 180,E1 -7806.391,E2 -7806.391} C_VEL
LIN {X 0,Y 469.363,Z 510.967,A -85,B 0,C 180,E1 -7806.434,E2 -7806.434} C_VEL
LIN {X 0,Y 469.244,Z 512.964,A -85,B 0,C 180,E1 -7806.461,E2 -7806.461} C_VEL
LIN {X 0,Y 467.567,Z 640.518,A -85,B 0,C 180,E1 -7808.48,E2 -7808.48} C_VEL
LIN {X 0,Y 467.112,Z 656.132,A -85,B 0,C 180,E1 -7808.896,E2 -7808.896} C_VEL
LIN {X 0,Y 466.48,Z 670.888,A -85,B 0,C 180,E1 -7809.465,E2 -7809.465} C_VEL
LIN {X 0,Y 465.752,Z 684.446,A -85,B 0,C 180,E1 -7810.154,E2 -7810.154} C_VEL
LIN {X 0,Y 464.882,Z 698.198,A -85,B 0,C 180,E1 -7811.034,E2 -7811.034} C_VEL
LIN {X 0,Y 463.916,Z 712.094,A -85,B 0,C 180,E1 -7812.137,E2 -7812.137} C_VEL
LIN {X 0,Y 463.071,Z 724.636,A -85,B 0,C 180,E1 -7813.355,E2 -7813.355} C_VEL
LIN {X 0,Y 462.239,Z 735.156,A -85,B 0,C 180,E1 -7814.571,E2 -7814.571} C_VEL
LIN {X 0,Y 461.429,Z 746.365,A -85,B 0,C 180,E1 -7816.122,E2 -7816.122} C_VEL
LIN {X 0,Y 460.858,Z 755.654,A -85,B 0,C 180,E1 -7817.674,E2 -7817.674} C_VEL
LIN {X 0,Y 460.483,Z 762.39,A -85,B 0,C 180,E1 -7819.003,E2 -7819.003} C_VEL
LIN {X 0,Y 460.008,Z 769.801,A -85,B 0,C 180,E1 -7820.77,E2 -7820.77} C_VEL
LIN {X 0,Y 459.771,Z 775.688,A -85,B 0,C 180,E1 -7822.536,E2 -7822.536} C_VEL
LIN {X 0,Y 459.637,Z 779.16,A -85,B 0,C 180,E1 -7823.857,E2 -7823.857} C_VEL
LIN {X 0,Y 459.535,Z 782.701,A -85,B 0,C 180,E1 -7825.616,E2 -7825.616} C_VEL
LIN {X 0,Y 459.561,Z 785.042,A -85,B 0,C 180,E1 -7827.372,E2 -7827.372} C_VEL
LIN {X 0,Y 459.492,Z 786.236,A -85,B 0,C 180,E1 -7829.125,E2 -7829.125} C_VEL
LIN {X 0,Y 459.492,Z 786.253,A -85,B 0,C 180,E1 -7830.878,E2 -7830.878} C_VEL
LIN {X 0,Y 459.562,Z 785.125,A -85,B 0,C 180,E1 -7832.631,E2 -7832.631} C_VEL
LIN {X 0,Y 459.535,Z 782.848,A -85,B 0,C 180,E1 -7834.387,E2 -7834.387} C_VEL
LIN {X 0,Y 459.649,Z 779.368,A -85,B 0,C 180,E1 -7836.145,E2 -7836.145} C_VEL
LIN {X 0,Y 459.817,Z 774.606,A -85,B 0,C 180,E1 -7837.908,E2 -7837.908} C_VEL
LIN {X 0,Y 460.078,Z 768.44,A -85,B 0,C 180,E1 -7839.675,E2 -7839.675} C_VEL
LIN {X 0,Y 460.592,Z 760.684,A -85,B 0,C 180,E1 -7841.442,E2 -7841.442} C_VEL
LIN {X 0,Y 461.017,Z 752.465,A -85,B 0,C 180,E1 -7842.987,E2 -7842.987} C_VEL
LIN {X 0,Y 461.719,Z 742.452,A -85,B 0,C 180,E1 -7844.547,E2 -7844.547} C_VEL
LIN {X 0,Y 462.428,Z 732.287,A -85,B 0,C 180,E1 -7845.878,E2 -7845.878} C_VEL
LIN {X 0,Y 463.346,Z 720.76,A -85,B 0,C 180,E1 -7847.141,E2 -7847.141} C_VEL
LIN {X 0,Y 464.234,Z 707.966,A -85,B 0,C 180,E1 -7848.31,E2 -7848.31} C_VEL
LIN {X 0,Y 465.09,Z 694.731,A -85,B 0,C 180,E1 -7849.304,E2 -7849.304} C_VEL
LIN {X 0,Y 466.028,Z 680.039,A -85,B 0,C 180,E1 -7850.181,E2 -7850.181} C_VEL
LIN {X 0,Y 466.72,Z 665.328,A -85,B 0,C 180,E1 -7850.865,E2 -7850.865} C_VEL
LIN {X 0,Y 467.345,Z 650.785,A -85,B 0,C 180,E1 -7851.36,E2 -7851.36} C_VEL
LIN {X 0,Y 467.705,Z 636.546,A -85,B 0,C 180,E1 -7851.69,E2 -7851.69} C_VEL
LIN {X 0,Y 469.446,Z 493.425,A -85,B 0,C 180,E1 -7853.942,E2 -7853.942} C_VEL
LIN {X 0,Y 465.931,Z 472.071,A -85,B 0,C 180,E1 -7854.509,E2 -7854.509} C_VEL
LIN {X 0,Y 466.767,Z 448.136,A -85,B 0,C 180,E1 -7857.027,E2 -7857.027} C_VEL
LIN {X 0,Y 468.016,Z 421.702,A -85,B 0,C 180,E1 -7859.955,E2 -7859.955} C_VEL
LIN {X 0,Y 468.944,Z 403.482,A -85,B 0,C 180,E1 -7861.997,E2 -7861.997} C_VEL
LIN {X 0,Y 467.369,Z 396.732,A -85,B 0,C 180,E1 -7862.89,E2 -7862.89} C_VEL
LIN {X 0,Y 462.129,Z 379.159,A -85,B 0,C 180,E1 -7865.304,E2 -7865.304} C_VEL
LIN {X 0,Y 460.491,Z 373.923,A -85,B 0,C 180,E1 -7866.08,E2 -7866.08} C_VEL
LIN {X 0,Y 460.482,Z 373.743,A -85,B 0,C 180,E1 -7868.888,E2 -7868.888} C_VEL
LIN {X 0,Y 460.498,Z 373.738,A -85,B 0,C 180,E1 -7871.598,E2 -7871.598} C_VEL
LIN {X 0,Y 460.505,Z 373.745,A -85,B 0,C 180,E1 -7874.591,E2 -7874.591} C_VEL
LIN {X 0,Y 460.475,Z 373.75,A -85,B 0,C 180,E1 -7877.813,E2 -7877.813} C_VEL
LIN {X 0,Y 460.485,Z 373.741,A -85,B 0,C 180,E1 -7881.113,E2 -7881.113} C_VEL
LIN {X 0,Y 460.502,Z 373.734,A -85,B 0,C 180,E1 -7884.553,E2 -7884.553} C_VEL
LIN {X 0,Y 460.502,Z 373.747,A -85,B 0,C 180,E1 -7887.713,E2 -7887.713} C_VEL
LIN {X 0,Y 460.519,Z 373.747,A -85,B 0,C 180,E1 -7890.767,E2 -7890.767} C_VEL
LIN {X 0,Y 460.526,Z 373.744,A -85,B 0,C 180,E1 -7894.211,E2 -7894.211} C_VEL
LIN {X 0,Y 460.552,Z 373.885,A -85,B 0,C 180,E1 -7897.366,E2 -7897.366} C_VEL
LIN {X 0,Y 462.521,Z 382.765,A -85,B 0,C 180,E1 -7899.101,E2 -7899.101} C_VEL
LIN {X 0,Y 465.75,Z 392.64,A -85,B 0,C 180,E1 -7899.464,E2 -7899.464} C_VEL
LIN {X 0,Y 466.94,Z 398.729,A -85,B 0,C 180,E1 -7899.631,E2 -7899.631} C_VEL
LIN {X 0,Y 465.073,Z 522.712,A -85,B 0,C 180,E1 -7901.842,E2 -7901.842} C_VEL
LIN {X 0,Y 464.873,Z 537.278,A -85,B 0,C 180,E1 -7902.278,E2 -7902.278} C_VEL
LIN {X 0,Y 464.555,Z 550.894,A -85,B 0,C 180,E1 -7902.854,E2 -7902.854} C_VEL
LIN {X 0,Y 464.093,Z 564.65,A -85,B 0,C 180,E1 -7903.617,E2 -7903.617} C_VEL
LIN {X 0,Y 463.615,Z 575.796,A -85,B 0,C 180,E1 -7904.391,E2 -7904.391} C_VEL
LIN {X 0,Y 463.135,Z 587.588,A -85,B 0,C 180,E1 -7905.387,E2 -7905.387} C_VEL
LIN {X 0,Y 462.576,Z 598.505,A -85,B 0,C 180,E1 -7906.501,E2 -7906.501} C_VEL
LIN {X 0,Y 462.101,Z 608.319,A -85,B 0,C 180,E1 -7907.706,E2 -7907.706} C_VEL
LIN {X 0,Y 461.632,Z 617.308,A -85,B 0,C 180,E1 -7909.029,E2 -7909.029} C_VEL
LIN {X 0,Y 461.239,Z 625.925,A -85,B 0,C 180,E1 -7910.572,E2 -7910.572} C_VEL
LIN {X 0,Y 460.921,Z 632.832,A -85,B 0,C 180,E1 -7912.112,E2 -7912.112} C_VEL
LIN {X 0,Y 460.759,Z 637.594,A -85,B 0,C 180,E1 -7913.431,E2 -7913.431} C_VEL
LIN {X 0,Y 460.509,Z 642.55,A -85,B 0,C 180,E1 -7915.185,E2 -7915.185} C_VEL
LIN {X 0,Y 460.341,Z 645.232,A -85,B 0,C 180,E1 -7916.499,E2 -7916.499} C_VEL
LIN {X 0,Y 460.425,Z 646.574,A -85,B 0,C 180,E1 -7917.375,E2 -7917.375} C_VEL
LIN {X 0,Y 460.379,Z 648.26,A -85,B 0,C 180,E1 -7919.125,E2 -7919.125} C_VEL
LIN {X 0,Y 460.385,Z 648.583,A -85,B 0,C 180,E1 -7920.875,E2 -7920.875} C_VEL
LIN {X 0,Y 460.508,Z 647.508,A -85,B 0,C 180,E1 -7922.624,E2 -7922.624} C_VEL
LIN {X 0,Y 460.576,Z 645.058,A -85,B 0,C 180,E1 -7924.376,E2 -7924.376} C_VEL
LIN {X 0,Y 460.911,Z 641.128,A -85,B 0,C 180,E1 -7926.127,E2 -7926.127} C_VEL
LIN {X 0,Y 461.169,Z 636.928,A -85,B 0,C 180,E1 -7927.515,E2 -7927.515} C_VEL
LIN {X 0,Y 461.51,Z 630.343,A -85,B 0,C 180,E1 -7929.201,E2 -7929.201} C_VEL
LIN {X 0,Y 462.018,Z 622.697,A -85,B 0,C 180,E1 -7930.739,E2 -7930.739} C_VEL
LIN {X 0,Y 462.529,Z 614.638,A -85,B 0,C 180,E1 -7932.059,E2 -7932.059} C_VEL
LIN {X 0,Y 463.109,Z 605.017,A -85,B 0,C 180,E1 -7933.362,E2 -7933.362} C_VEL
LIN {X 0,Y 463.725,Z 593.95,A -85,B 0,C 180,E1 -7934.593,E2 -7934.593} C_VEL
LIN {X 0,Y 464.333,Z 581.744,A -85,B 0,C 180,E1 -7935.697,E2 -7935.697} C_VEL
LIN {X 0,Y 464.761,Z 569.704,A -85,B 0,C 180,E1 -7936.584,E2 -7936.584} C_VEL
LIN {X 0,Y 465.29,Z 556.407,A -85,B 0,C 180,E1 -7937.356,E2 -7937.356} C_VEL
LIN {X 0,Y 465.676,Z 542.86,A -85,B 0,C 180,E1 -7937.959,E2 -7937.959} C_VEL
LIN {X 0,Y 465.805,Z 528.508,A -85,B 0,C 180,E1 -7938.423,E2 -7938.423} C_VEL
LIN {X 0,Y 468.175,Z 433.155,A -85,B 0,C 180,E1 -7940.39,E2 -7940.39} C_VEL
LIN {X 0,Y 469.128,Z 400.286,A -85,B 0,C 180,E1 -7941.109,E2 -7941.109} C_VEL
LIN {X 0,Y 467.346,Z 395.747,A -85,B 0,C 180,E1 -7941.341,E2 -7941.341} C_VEL
LIN {X 0,Y 465.396,Z 391.678,A -85,B 0,C 180,E1 -7941.601,E2 -7941.601} C_VEL
LIN {X 0,Y 462.628,Z 380.886,A -85,B 0,C 180,E1 -7944.287,E2 -7944.287} C_VEL
LIN {X 0,Y 460.568,Z 373.805,A -85,B 0,C 180,E1 -7946.265,E2 -7946.265} C_VEL
LIN {X 0,Y 460.545,Z 373.745,A -85,B 0,C 180,E1 -7949.231,E2 -7949.231} C_VEL
LIN {X 0,Y 460.536,Z 373.747,A -85,B 0,C 180,E1 -7952.284,E2 -7952.284} C_VEL
LIN {X 0,Y 460.513,Z 373.747,A -85,B 0,C 180,E1 -7955.445,E2 -7955.445} C_VEL
LIN {X 0,Y 460.535,Z 373.745,A -85,B 0,C 180,E1 -7958.895,E2 -7958.895} C_VEL
LIN {X 0,Y 460.508,Z 373.749,A -85,B 0,C 180,E1 -7962.183,E2 -7962.183} C_VEL
LIN {X 0,Y 460.515,Z 373.747,A -85,B 0,C 180,E1 -7965.41,E2 -7965.41} C_VEL
LIN {X 0,Y 460.519,Z 373.748,A -85,B 0,C 180,E1 -7968.986,E2 -7968.986} C_VEL
LIN {X 0,Y 460.486,Z 373.753,A -85,B 0,C 180,E1 -7972.374,E2 -7972.374} C_VEL
LIN {X 0,Y 460.554,Z 373.979,A -85,B 0,C 180,E1 -7974.088,E2 -7974.088} C_VEL
LIN {X 0,Y 463.471,Z 382.381,A -85,B 0,C 180,E1 -7975.709,E2 -7975.709} C_VEL
LIN {X 0,Y 466.711,Z 393.057,A -85,B 0,C 180,E1 -7977.488,E2 -7977.488} C_VEL
LIN {X 0,Y 468.65,Z 401.437,A -85,B 0,C 180,E1 -7978.736,E2 -7978.736} C_VEL
LIN {X 0,Y 467.787,Z 413.325,A -85,B 0,C 180,E1 -7980.153,E2 -7980.153} C_VEL
LIN {X 0,Y 465.894,Z 440.306,A -85,B 0,C 180,E1 -7983.213,E2 -7983.213} C_VEL
LIN {X 0,Y 464.811,Z 461.211,A -85,B 0,C 180,E1 -7985.49,E2 -7985.49} C_VEL
LIN {X 0,Y 467.132,Z 479.341,A -85,B 0,C 180,E1 -7986.019,E2 -7986.019} C_VEL
LIN {X 0,Y 468.711,Z 493.534,A -85,B 0,C 180,E1 -7986.337,E2 -7986.337} C_VEL
LIN {X 0,Y 466.983,Z 640.155,A -85,B 0,C 180,E1 -7988.652,E2 -7988.652} C_VEL
LIN {X 0,Y 466.589,Z 654.392,A -85,B 0,C 180,E1 -7989.023,E2 -7989.023} C_VEL
LIN {X 0,Y 466.049,Z 668.069,A -85,B 0,C 180,E1 -7989.531,E2 -7989.531} C_VEL
LIN {X 0,Y 465.322,Z 682.615,A -85,B 0,C 180,E1 -7990.247,E2 -7990.247} C_VEL
LIN {X 0,Y 464.545,Z 696.602,A -85,B 0,C 180,E1 -7991.132,E2 -7991.132} C_VEL
LIN {X 0,Y 463.698,Z 709.353,A -85,B 0,C 180,E1 -7992.125,E2 -7992.125} C_VEL
LIN {X 0,Y 462.805,Z 722.197,A -85,B 0,C 180,E1 -7993.343,E2 -7993.343} C_VEL
LIN {X 0,Y 462.065,Z 732.923,A -85,B 0,C 180,E1 -7994.562,E2 -7994.562} C_VEL
LIN {X 0,Y 461.421,Z 742.819,A -85,B 0,C 180,E1 -7995.894,E2 -7995.894} C_VEL
LIN {X 0,Y 460.73,Z 752.728,A -85,B 0,C 180,E1 -7997.49,E2 -7997.49} C_VEL
LIN {X 0,Y 460.409,Z 760.507,A -85,B 0,C 180,E1 -7998.999,E2 -7998.999} C_VEL
LIN {X 0,Y 460.001,Z 767.976,A -85,B 0,C 180,E1 -8000.767,E2 -8000.767} C_VEL
LIN {X 0,Y 459.788,Z 773.893,A -85,B 0,C 180,E1 -8002.533,E2 -8002.533} C_VEL
LIN {X 0,Y 459.717,Z 777.389,A -85,B 0,C 180,E1 -8003.856,E2 -8003.856} C_VEL
LIN {X 0,Y 459.626,Z 780.943,A -85,B 0,C 180,E1 -8005.614,E2 -8005.614} C_VEL
LIN {X 0,Y 459.641,Z 783.277,A -85,B 0,C 180,E1 -8007.37,E2 -8007.37} C_VEL
LIN {X 0,Y 459.573,Z 784.45,A -85,B 0,C 180,E1 -8009.122,E2 -8009.122} C_VEL
LIN {X 0,Y 459.573,Z 784.45,A -85,B 0,C 180,E1 -8010.875,E2 -8010.875} C_VEL
LIN {X 0,Y 459.641,Z 783.276,A -85,B 0,C 180,E1 -8012.628,E2 -8012.628} C_VEL
LIN {X 0,Y 459.607,Z 780.942,A -85,B 0,C 180,E1 -8014.384,E2 -8014.384} C_VEL
LIN {X 0,Y 459.695,Z 777.397,A -85,B 0,C 180,E1 -8016.142,E2 -8016.142} C_VEL
LIN {X 0,Y 459.829,Z 772.547,A -85,B 0,C 180,E1 -8017.905,E2 -8017.905} C_VEL
LIN {X 0,Y 460.074,Z 766.258,A -85,B 0,C 180,E1 -8019.672,E2 -8019.672} C_VEL
LIN {X 0,Y 460.519,Z 758.353,A -85,B 0,C 180,E1 -8021.442,E2 -8021.442} C_VEL
LIN {X 0,Y 460.92,Z 750.044,A -85,B 0,C 180,E1 -8022.973,E2 -8022.973} C_VEL
LIN {X 0,Y 461.493,Z 741.335,A -85,B 0,C 180,E1 -8024.326,E2 -8024.326} C_VEL
LIN {X 0,Y 462.156,Z 731.163,A -85,B 0,C 180,E1 -8025.658,E2 -8025.658} C_VEL
LIN {X 0,Y 463.021,Z 718.789,A -85,B 0,C 180,E1 -8027.011,E2 -8027.011} C_VEL
LIN {X 0,Y 463.928,Z 705.443,A -85,B 0,C 180,E1 -8028.205,E2 -8028.205} C_VEL
LIN {X 0,Y 464.769,Z 691.783,A -85,B 0,C 180,E1 -8029.2,E2 -8029.2} C_VEL
LIN {X 0,Y 465.568,Z 677.555,A -85,B 0,C 180,E1 -8030.026,E2 -8030.026} C_VEL
LIN {X 0,Y 466.228,Z 663.054,A -85,B 0,C 180,E1 -8030.677,E2 -8030.677} C_VEL
LIN {X 0,Y 466.727,Z 648.539,A -85,B 0,C 180,E1 -8031.152,E2 -8031.152} C_VEL
LIN {X 0,Y 467.069,Z 632.578,A -85,B 0,C 180,E1 -8031.486,E2 -8031.486} C_VEL
LIN {X 0,Y 468.698,Z 492.985,A -85,B 0,C 180,E1 -8033.67,E2 -8033.67} C_VEL
LIN {X 0,Y 465.087,Z 465.477,A -85,B 0,C 180,E1 -8034.341,E2 -8034.341} C_VEL
LIN {X 0,Y 466.619,Z 435.958,A -85,B 0,C 180,E1 -8037.473,E2 -8037.473} C_VEL
LIN {X 0,Y 468.271,Z 407.502,A -85,B 0,C 180,E1 -8040.556,E2 -8040.556} C_VEL
LIN {X 0,Y 468.493,Z 401.416,A -85,B 0,C 180,E1 -8041.232,E2 -8041.232} C_VEL
LIN {X 0,Y 463.606,Z 384.208,A -85,B 0,C 180,E1 -8043.512,E2 -8043.512} C_VEL
LIN {X 0,Y 460.542,Z 373.92,A -85,B 0,C 180,E1 -8044.971,E2 -8044.971} C_VEL
LIN {X 0,Y 460.49,Z 373.751,A -85,B 0,C 180,E1 -8048.734,E2 -8048.734} C_VEL
LIN {X 0,Y 460.496,Z 373.748,A -85,B 0,C 180,E1 -8051.597,E2 -8051.597} C_VEL
LIN {X 0,Y 460.499,Z 373.75,A -85,B 0,C 180,E1 -8054.588,E2 -8054.588} C_VEL
LIN {X 0,Y 460.46,Z 373.728,A -85,B 0,C 180,E1 -8057.812,E2 -8057.812} C_VEL
LIN {X 0,Y 460.497,Z 373.744,A -85,B 0,C 180,E1 -8060.134,E2 -8060.134} C_VEL
LIN {X 0,Y 460.445,Z 373.74,A -85,B 0,C 180,E1 -8063.468,E2 -8063.468} C_VEL
LIN {X 0,Y 460.502,Z 373.737,A -85,B 0,C 180,E1 -8066.673,E2 -8066.673} C_VEL
LIN {X 0,Y 460.489,Z 373.747,A -85,B 0,C 180,E1 -8069.758,E2 -8069.758} C_VEL
LIN {X 0,Y 460.477,Z 373.751,A -85,B 0,C 180,E1 -8072.75,E2 -8072.75} C_VEL
LIN {X 0,Y 460.505,Z 373.736,A -85,B 0,C 180,E1 -8075.666,E2 -8075.666} C_VEL
LIN {X 0,Y 460.506,Z 373.745,A -85,B 0,C 180,E1 -8078.578,E2 -8078.578} C_VEL
LIN {X 0,Y 460.566,Z 373.735,A -85,B 0,C 180,E1 -8081.31,E2 -8081.31} C_VEL
LIN {X 0,Y 460.531,Z 373.733,A -85,B 0,C 180,E1 -8084.964,E2 -8084.964} C_VEL
LIN {X 0,Y 460.589,Z 373.736,A -85,B 0,C 180,E1 -8088.559,E2 -8088.559} C_VEL
LIN {X 0,Y 460.606,Z 373.729,A -85,B 0,C 180,E1 -8092.107,E2 -8092.107} C_VEL
LIN {X 0,Y 460.651,Z 373.721,A -85,B 0,C 180,E1 -8094.748,E2 -8094.748} C_VEL
LIN {X 0,Y 460.749,Z 373.712,A -85,B 0,C 180,E1 -8097.377,E2 -8097.377} C_VEL
LIN {X 0,Y 460.779,Z 373.71,A -85,B 0,C 180,E1 -8100,E2 -8100} C_VEL
LIN {X 0,Y 460.745,Z 373.714,A -85,B 0,C 180,E1 -8102.623,E2 -8102.623} C_VEL
LIN {X 0,Y 460.67,Z 373.721,A -85,B 0,C 180,E1 -8106.131,E2 -8106.131} C_VEL
LIN {X 0,Y 460.592,Z 373.738,A -85,B 0,C 180,E1 -8108.777,E2 -8108.777} C_VEL
LIN {X 0,Y 460.581,Z 373.728,A -85,B 0,C 180,E1 -8112.436,E2 -8112.436} C_VEL
LIN {X 0,Y 460.585,Z 373.73,A -85,B 0,C 180,E1 -8115.998,E2 -8115.998} C_VEL
LIN {X 0,Y 460.552,Z 373.737,A -85,B 0,C 180,E1 -8119.616,E2 -8119.616} C_VEL
LIN {X 0,Y 460.492,Z 373.745,A -85,B 0,C 180,E1 -8122.43,E2 -8122.43} C_VEL
LIN {X 0,Y 460.508,Z 373.738,A -85,B 0,C 180,E1 -8125.791,E2 -8125.791} C_VEL
LIN {X 0,Y 460.5,Z 373.743,A -85,B 0,C 180,E1 -8129.234,E2 -8129.234} C_VEL
LIN {X 0,Y 460.501,Z 373.748,A -85,B 0,C 180,E1 -8132.287,E2 -8132.287} C_VEL
LIN {X 0,Y 460.492,Z 373.745,A -85,B 0,C 180,E1 -8135.447,E2 -8135.447} C_VEL
LIN {X 0,Y 460.48,Z 373.742,A -85,B 0,C 180,E1 -8138.891,E2 -8138.891} C_VEL
LIN {X 0,Y 460.489,Z 373.74,A -85,B 0,C 180,E1 -8141.599,E2 -8141.599} C_VEL
LIN {X 0,Y 460.494,Z 373.75,A -85,B 0,C 180,E1 -8144.591,E2 -8144.591} C_VEL
LIN {X 0,Y 460.463,Z 373.751,A -85,B 0,C 180,E1 -8147.814,E2 -8147.814} C_VEL
LIN {X 0,Y 460.5,Z 373.738,A -85,B 0,C 180,E1 -8150.137,E2 -8150.137} C_VEL
LIN {X 0,Y 460.451,Z 373.747,A -85,B 0,C 180,E1 -8153.47,E2 -8153.47} C_VEL
LIN {X 0,Y 460.53,Z 373.935,A -85,B 0,C 180,E1 -8154.028,E2 -8154.028} C_VEL
LIN {X 0,Y 465.629,Z 390.442,A -85,B 0,C 180,E1 -8156.365,E2 -8156.365} C_VEL
LIN {X 0,Y 468.928,Z 402.82,A -85,B 0,C 180,E1 -8158.017,E2 -8158.017} C_VEL
LIN {X 0,Y 467.631,Z 430.258,A -85,B 0,C 180,E1 -8161.102,E2 -8161.102} C_VEL
LIN {X 0,Y 466.285,Z 461.7,A -85,B 0,C 180,E1 -8164.52,E2 -8164.52} C_VEL
LIN {X 0,Y 465.966,Z 472.345,A -85,B 0,C 180,E1 -8165.6,E2 -8165.6} C_VEL
LIN {X 0,Y 469.48,Z 493.992,A -85,B 0,C 180,E1 -8166.162,E2 -8166.162} C_VEL
LIN {X 0,Y 469.244,Z 512.964,A -85,B 0,C 180,E1 -8166.461,E2 -8166.461} C_VEL
LIN {X 0,Y 468.509,Z 518.816,A -85,B 0,C 180,E1 -8166.518,E2 -8166.518} C_VEL
LIN {X 0,Y 462.993,Z 537.874,A -85,B 0,C 180,E1 -8166.539,E2 -8166.539} C_VEL
LIN {X 0,Y 462.349,Z 543.721,A -85,B 0,C 180,E1 -8166.602,E2 -8166.602} C_VEL
LIN {X 0,Y 460.978,Z 640.424,A -85,B 0,C 180,E1 -8168.157,E2 -8168.157} C_VEL
LIN {X 0,Y 460.527,Z 656.013,A -85,B 0,C 180,E1 -8168.577,E2 -8168.577} C_VEL
LIN {X 0,Y 459.894,Z 669.497,A -85,B 0,C 180,E1 -8169.094,E2 -8169.094} C_VEL
LIN {X 0,Y 459.049,Z 684.411,A -85,B 0,C 180,E1 -8169.852,E2 -8169.852} C_VEL
LIN {X 0,Y 458.139,Z 698.17,A -85,B 0,C 180,E1 -8170.744,E2 -8170.744} C_VEL
LIN {X 0,Y 457.13,Z 712.07,A -85,B 0,C 180,E1 -8171.862,E2 -8171.862} C_VEL
LIN {X 0,Y 456.218,Z 724.615,A -85,B 0,C 180,E1 -8173.098,E2 -8173.098} C_VEL
LIN {X 0,Y 455.352,Z 735.136,A -85,B 0,C 180,E1 -8174.331,E2 -8174.331} C_VEL
LIN {X 0,Y 454.479,Z 746.348,A -85,B 0,C 180,E1 -8175.905,E2 -8175.905} C_VEL
LIN {X 0,Y 453.869,Z 755.638,A -85,B 0,C 180,E1 -8177.481,E2 -8177.481} C_VEL
LIN {X 0,Y 453.456,Z 762.374,A -85,B 0,C 180,E1 -8178.831,E2 -8178.831} C_VEL
LIN {X 0,Y 452.964,Z 769.786,A -85,B 0,C 180,E1 -8180.625,E2 -8180.625} C_VEL
LIN {X 0,Y 452.697,Z 775.674,A -85,B 0,C 180,E1 -8182.419,E2 -8182.419} C_VEL
LIN {X 0,Y 452.562,Z 779.146,A -85,B 0,C 180,E1 -8183.761,E2 -8183.761} C_VEL
LIN {X 0,Y 452.454,Z 782.687,A -85,B 0,C 180,E1 -8185.547,E2 -8185.547} C_VEL
LIN {X 0,Y 452.484,Z 785.029,A -85,B 0,C 180,E1 -8187.331,E2 -8187.331} C_VEL
LIN {X 0,Y 452.4,Z 786.223,A -85,B 0,C 180,E1 -8189.111,E2 -8189.111} C_VEL
LIN {X 0,Y 452.401,Z 786.239,A -85,B 0,C 180,E1 -8190.891,E2 -8190.891} C_VEL
LIN {X 0,Y 452.486,Z 785.11,A -85,B 0,C 180,E1 -8192.672,E2 -8192.672} C_VEL
LIN {X 0,Y 452.454,Z 782.832,A -85,B 0,C 180,E1 -8194.456,E2 -8194.456} C_VEL
LIN {X 0,Y 452.602,Z 779.007,A -85,B 0,C 180,E1 -8196.388,E2 -8196.388} C_VEL
LIN {X 0,Y 452.742,Z 774.588,A -85,B 0,C 180,E1 -8198.032,E2 -8198.032} C_VEL
LIN {X 0,Y 453.012,Z 768.42,A -85,B 0,C 180,E1 -8199.827,E2 -8199.827} C_VEL
LIN {X 0,Y 453.574,Z 760.663,A -85,B 0,C 180,E1 -8201.622,E2 -8201.622} C_VEL
LIN {X 0,Y 454.021,Z 752.523,A -85,B 0,C 180,E1 -8203.177,E2 -8203.177} C_VEL
LIN {X 0,Y 454.792,Z 742.427,A -85,B 0,C 180,E1 -8204.773,E2 -8204.773} C_VEL
LIN {X 0,Y 455.559,Z 732.259,A -85,B 0,C 180,E1 -8206.124,E2 -8206.124} C_VEL
LIN {X 0,Y 456.559,Z 720.045,A -85,B 0,C 180,E1 -8207.473,E2 -8207.473} C_VEL
LIN {X 0,Y 457.457,Z 707.929,A -85,B 0,C 180,E1 -8208.591,E2 -8208.591} C_VEL
LIN {X 0,Y 458.35,Z 694.686,A -85,B 0,C 180,E1 -8209.599,E2 -8209.599} C_VEL
LIN {X 0,Y 459.283,Z 681.057,A -85,B 0,C 180,E1 -8210.432,E2 -8210.432} C_VEL
LIN {X 0,Y 460.07,Z 665.74,A -85,B 0,C 180,E1 -8211.161,E2 -8211.161} C_VEL
LIN {X 0,Y 460.747,Z 650.68,A -85,B 0,C 180,E1 -8211.681,E2 -8211.681} C_VEL
LIN {X 0,Y 461.118,Z 636.392,A -85,B 0,C 180,E1 -8212.016,E2 -8212.016} C_VEL
LIN {X 0,Y 462.987,Z 494.877,A -85,B 0,C 180,E1 -8214.27,E2 -8214.27} C_VEL
LIN {X 0,Y 459.257,Z 471.986,A -85,B 0,C 180,E1 -8214.889,E2 -8214.889} C_VEL
LIN {X 0,Y 460.165,Z 448.435,A -85,B 0,C 180,E1 -8217.387,E2 -8217.387} C_VEL
LIN {X 0,Y 461.625,Z 419.093,A -85,B 0,C 180,E1 -8220.666,E2 -8220.666} C_VEL
LIN {X 0,Y 462.262,Z 404.516,A -85,B 0,C 180,E1 -8222.332,E2 -8222.332} C_VEL
LIN {X 0,Y 457.512,Z 387.793,A -85,B 0,C 180,E1 -8224.638,E2 -8224.638} C_VEL
LIN {X 0,Y 453.438,Z 374.825,A -85,B 0,C 180,E1 -8226.517,E2 -8226.517} C_VEL
LIN {X 0,Y 453.422,Z 374.623,A -85,B 0,C 180,E1 -8229.458,E2 -8229.458} C_VEL
LIN {X 0,Y 453.434,Z 374.616,A -85,B 0,C 180,E1 -8231.929,E2 -8231.929} C_VEL
LIN {X 0,Y 453.471,Z 374.611,A -85,B 0,C 180,E1 -8235.474,E2 -8235.474} C_VEL
LIN {X 0,Y 453.44,Z 374.626,A -85,B 0,C 180,E1 -8238.205,E2 -8238.205} C_VEL
LIN {X 0,Y 453.428,Z 374.615,A -85,B 0,C 180,E1 -8240.805,E2 -8240.805} C_VEL
LIN {X 0,Y 453.444,Z 374.617,A -85,B 0,C 180,E1 -8243.916,E2 -8243.916} C_VEL
LIN {X 0,Y 453.469,Z 374.614,A -85,B 0,C 180,E1 -8246.816,E2 -8246.816} C_VEL
LIN {X 0,Y 453.458,Z 374.624,A -85,B 0,C 180,E1 -8250.267,E2 -8250.267} C_VEL
LIN {X 0,Y 453.427,Z 374.632,A -85,B 0,C 180,E1 -8253.289,E2 -8253.289} C_VEL
LIN {X 0,Y 453.495,Z 374.621,A -85,B 0,C 180,E1 -8256.238,E2 -8256.238} C_VEL
LIN {X 0,Y 453.547,Z 374.805,A -85,B 0,C 180,E1 -8257.117,E2 -8257.117} C_VEL
LIN {X 0,Y 455.463,Z 383.436,A -85,B 0,C 180,E1 -8258.8,E2 -8258.8} C_VEL
LIN {X 0,Y 459.265,Z 394.616,A -85,B 0,C 180,E1 -8259.209,E2 -8259.209} C_VEL
LIN {X 0,Y 460.242,Z 399.358,A -85,B 0,C 180,E1 -8259.344,E2 -8259.344} C_VEL
LIN {X 0,Y 458.23,Z 523.85,A -85,B 0,C 180,E1 -8261.617,E2 -8261.617} C_VEL
LIN {X 0,Y 458.047,Z 538.408,A -85,B 0,C 180,E1 -8262.066,E2 -8262.066} C_VEL
LIN {X 0,Y 457.702,Z 552.294,A -85,B 0,C 180,E1 -8262.668,E2 -8262.668} C_VEL
LIN {X 0,Y 457.202,Z 566.498,A -85,B 0,C 180,E1 -8263.478,E2 -8263.478} C_VEL
LIN {X 0,Y 456.697,Z 578.918,A -85,B 0,C 180,E1 -8264.377,E2 -8264.377} C_VEL
LIN {X 0,Y 456.085,Z 591.465,A -85,B 0,C 180,E1 -8265.499,E2 -8265.499} C_VEL
LIN {X 0,Y 455.55,Z 601.809,A -85,B 0,C 180,E1 -8266.62,E2 -8266.62} C_VEL
LIN {X 0,Y 455.014,Z 612.085,A -85,B 0,C 180,E1 -8267.964,E2 -8267.964} C_VEL
LIN {X 0,Y 454.539,Z 620.611,A -85,B 0,C 180,E1 -8269.307,E2 -8269.307} C_VEL
LIN {X 0,Y 454.188,Z 628.763,A -85,B 0,C 180,E1 -8270.874,E2 -8270.874} C_VEL
LIN {X 0,Y 453.848,Z 634.955,A -85,B 0,C 180,E1 -8272.339,E2 -8272.339} C_VEL
LIN {X 0,Y 453.627,Z 639.838,A -85,B 0,C 180,E1 -8273.774,E2 -8273.774} C_VEL
LIN {X 0,Y 453.374,Z 644.45,A -85,B 0,C 180,E1 -8275.555,E2 -8275.555} C_VEL
LIN {X 0,Y 453.408,Z 647.555,A -85,B 0,C 180,E1 -8277.335,E2 -8277.335} C_VEL
LIN {X 0,Y 453.361,Z 649.283,A -85,B 0,C 180,E1 -8279.112,E2 -8279.112} C_VEL
LIN {X 0,Y 453.369,Z 649.649,A -85,B 0,C 180,E1 -8280.888,E2 -8280.888} C_VEL
LIN {X 0,Y 453.519,Z 648.614,A -85,B 0,C 180,E1 -8282.665,E2 -8282.665} C_VEL
LIN {X 0,Y 453.588,Z 646.205,A -85,B 0,C 180,E1 -8284.443,E2 -8284.443} C_VEL
LIN {X 0,Y 453.948,Z 642.303,A -85,B 0,C 180,E1 -8286.221,E2 -8286.221} C_VEL
LIN {X 0,Y 454.246,Z 637.974,A -85,B 0,C 180,E1 -8287.672,E2 -8287.672} C_VEL
LIN {X 0,Y 454.617,Z 631.537,A -85,B 0,C 180,E1 -8289.342,E2 -8289.342} C_VEL
LIN {X 0,Y 455.153,Z 623.895,A -85,B 0,C 180,E1 -8290.903,E2 -8290.903} C_VEL
LIN {X 0,Y 455.716,Z 615.868,A -85,B 0,C 180,E1 -8292.242,E2 -8292.242} C_VEL
LIN {X 0,Y 456.331,Z 606.159,A -85,B 0,C 180,E1 -8293.584,E2 -8293.584} C_VEL
LIN {X 0,Y 456.995,Z 595.309,A -85,B 0,C 180,E1 -8294.813,E2 -8294.813} C_VEL
LIN {X 0,Y 457.614,Z 583.135,A -85,B 0,C 180,E1 -8295.933,E2 -8295.933} C_VEL
LIN {X 0,Y 458.078,Z 571.135,A -85,B 0,C 180,E1 -8296.833,E2 -8296.833} C_VEL
LIN {X 0,Y 458.666,Z 556.875,A -85,B 0,C 180,E1 -8297.673,E2 -8297.673} C_VEL
LIN {X 0,Y 459.101,Z 542.526,A -85,B 0,C 180,E1 -8298.313,E2 -8298.313} C_VEL
LIN {X 0,Y 459.246,Z 529.003,A -85,B 0,C 180,E1 -8298.746,E2 -8298.746} C_VEL
LIN {X 0,Y 461.597,Z 442.649,A -85,B 0,C 180,E1 -8300.577,E2 -8300.577} C_VEL
LIN {X 0,Y 462.929,Z 401.988,A -85,B 0,C 180,E1 -8301.494,E2 -8301.494} C_VEL
LIN {X 0,Y 458.515,Z 392.91,A -85,B 0,C 180,E1 -8302.076,E2 -8302.076} C_VEL
LIN {X 0,Y 456.013,Z 383.087,A -85,B 0,C 180,E1 -8304.59,E2 -8304.59} C_VEL
LIN {X 0,Y 454.368,Z 377.344,A -85,B 0,C 180,E1 -8306.216,E2 -8306.216} C_VEL
LIN {X 0,Y 453.547,Z 374.66,A -85,B 0,C 180,E1 -8307.077,E2 -8307.077} C_VEL
LIN {X 0,Y 453.477,Z 374.625,A -85,B 0,C 180,E1 -8309.784,E2 -8309.784} C_VEL
LIN {X 0,Y 453.495,Z 374.622,A -85,B 0,C 180,E1 -8313.189,E2 -8313.189} C_VEL
LIN {X 0,Y 453.455,Z 374.628,A -85,B 0,C 180,E1 -8316.298,E2 -8316.298} C_VEL
LIN {X 0,Y 453.468,Z 374.624,A -85,B 0,C 180,E1 -8319.452,E2 -8319.452} C_VEL
LIN {X 0,Y 453.464,Z 374.628,A -85,B 0,C 180,E1 -8321.932,E2 -8321.932} C_VEL
LIN {X 0,Y 453.485,Z 374.623,A -85,B 0,C 180,E1 -8325.471,E2 -8325.471} C_VEL
LIN {X 0,Y 453.449,Z 374.63,A -85,B 0,C 180,E1 -8328.205,E2 -8328.205} C_VEL
LIN {X 0,Y 453.442,Z 374.629,A -85,B 0,C 180,E1 -8330.801,E2 -8330.801} C_VEL
LIN {X 0,Y 453.453,Z 374.853,A -85,B 0,C 180,E1 -8333.331,E2 -8333.331} C_VEL
LIN {X 0,Y 455.924,Z 381.695,A -85,B 0,C 180,E1 -8334.784,E2 -8334.784} C_VEL
LIN {X 0,Y 459.089,Z 391.379,A -85,B 0,C 180,E1 -8336.556,E2 -8336.556} C_VEL
LIN {X 0,Y 461.815,Z 401.926,A -85,B 0,C 180,E1 -8338.244,E2 -8338.244} C_VEL
LIN {X 0,Y 462.18,Z 405.144,A -85,B 0,C 180,E1 -8338.698,E2 -8338.698} C_VEL
LIN {X 0,Y 459.888,Z 431.736,A -85,B 0,C 180,E1 -8341.846,E2 -8341.846} C_VEL
LIN {X 0,Y 458.178,Z 458.031,A -85,B 0,C 180,E1 -8344.823,E2 -8344.823} C_VEL
LIN {X 0,Y 458.181,Z 460.848,A -85,B 0,C 180,E1 -8345.084,E2 -8345.084} C_VEL
LIN {X 0,Y 460.895,Z 482.552,A -85,B 0,C 180,E1 -8345.724,E2 -8345.724} C_VEL
LIN {X 0,Y 462.228,Z 493.689,A -85,B 0,C 180,E1 -8345.985,E2 -8345.985} C_VEL
LIN {X 0,Y 460.422,Z 638.812,A -85,B 0,C 180,E1 -8348.303,E2 -8348.303} C_VEL
LIN {X 0,Y 460.019,Z 653.637,A -85,B 0,C 180,E1 -8348.682,E2 -8348.682} C_VEL
LIN {X 0,Y 459.437,Z 667.219,A -85,B 0,C 180,E1 -8349.182,E2 -8349.182} C_VEL
LIN {X 0,Y 458.76,Z 680.685,A -85,B 0,C 180,E1 -8349.836,E2 -8349.836} C_VEL
LIN {X 0,Y 458.063,Z 693.492,A -85,B 0,C 180,E1 -8350.621,E2 -8350.621} C_VEL
LIN {X 0,Y 457.071,Z 706.815,A -85,B 0,C 180,E1 -8351.625,E2 -8351.625} C_VEL
LIN {X 0,Y 456.192,Z 719.296,A -85,B 0,C 180,E1 -8352.777,E2 -8352.777} C_VEL
LIN {X 0,Y 455.302,Z 731.171,A -85,B 0,C 180,E1 -8354.097,E2 -8354.097} C_VEL
LIN {X 0,Y 454.622,Z 741.343,A -85,B 0,C 180,E1 -8355.45,E2 -8355.45} C_VEL
LIN {X 0,Y 453.855,Z 751.514,A -85,B 0,C 180,E1 -8357.069,E2 -8357.069} C_VEL
LIN {X 0,Y 453.444,Z 759.479,A -85,B 0,C 180,E1 -8358.601,E2 -8358.601} C_VEL
LIN {X 0,Y 453.012,Z 766.27,A -85,B 0,C 180,E1 -8360.173,E2 -8360.173} C_VEL
LIN {X 0,Y 452.785,Z 772.552,A -85,B 0,C 180,E1 -8361.968,E2 -8361.968} C_VEL
LIN {X 0,Y 452.651,Z 777.405,A -85,B 0,C 180,E1 -8363.759,E2 -8363.759} C_VEL
LIN {X 0,Y 452.539,Z 780.957,A -85,B 0,C 180,E1 -8365.545,E2 -8365.545} C_VEL
LIN {X 0,Y 452.561,Z 783.292,A -85,B 0,C 180,E1 -8367.328,E2 -8367.328} C_VEL
LIN {X 0,Y 452.477,Z 784.464,A -85,B 0,C 180,E1 -8369.109,E2 -8369.109} C_VEL
LIN {X 0,Y 452.477,Z 784.464,A -85,B 0,C 180,E1 -8370.889,E2 -8370.889} C_VEL
LIN {X 0,Y 452.563,Z 783.29,A -85,B 0,C 180,E1 -8372.669,E2 -8372.669} C_VEL
LIN {X 0,Y 452.522,Z 780.957,A -85,B 0,C 180,E1 -8374.452,E2 -8374.452} C_VEL
LIN {X 0,Y 452.625,Z 776.994,A -85,B 0,C 180,E1 -8376.415,E2 -8376.415} C_VEL
LIN {X 0,Y 452.776,Z 772.562,A -85,B 0,C 180,E1 -8378.029,E2 -8378.029} C_VEL
LIN {X 0,Y 453.01,Z 766.275,A -85,B 0,C 180,E1 -8379.824,E2 -8379.824} C_VEL
LIN {X 0,Y 453.509,Z 758.37,A -85,B 0,C 180,E1 -8381.621,E2 -8381.621} C_VEL
LIN {X 0,Y 453.952,Z 750.063,A -85,B 0,C 180,E1 -8383.176,E2 -8383.176} C_VEL
LIN {X 0,Y 454.552,Z 741.355,A -85,B 0,C 180,E1 -8384.55,E2 -8384.55} C_VEL
LIN {X 0,Y 455.258,Z 731.185,A -85,B 0,C 180,E1 -8385.902,E2 -8385.902} C_VEL
LIN {X 0,Y 456.146,Z 719.482,A -85,B 0,C 180,E1 -8387.205,E2 -8387.205} C_VEL
LIN {X 0,Y 457.055,Z 706.835,A -85,B 0,C 180,E1 -8388.373,E2 -8388.373} C_VEL
LIN {X 0,Y 457.942,Z 693.501,A -85,B 0,C 180,E1 -8389.381,E2 -8389.381} C_VEL
LIN {X 0,Y 458.848,Z 678.706,A -85,B 0,C 180,E1 -8390.274,E2 -8390.274} C_VEL
LIN {X 0,Y 459.578,Z 663.682,A -85,B 0,C 180,E1 -8390.968,E2 -8390.968} C_VEL
LIN {X 0,Y 460.147,Z 648.057,A -85,B 0,C 180,E1 -8391.484,E2 -8391.484} C_VEL
LIN {X 0,Y 460.475,Z 632.715,A -85,B 0,C 180,E1 -8391.809,E2 -8391.809} C_VEL
LIN {X 0,Y 462.223,Z 493.634,A -85,B 0,C 180,E1 -8394.014,E2 -8394.014} C_VEL
LIN {X 0,Y 458.374,Z 465.095,A -85,B 0,C 180,E1 -8394.718,E2 -8394.718} C_VEL
LIN {X 0,Y 458.352,Z 463.032,A -85,B 0,C 180,E1 -8394.872,E2 -8394.872} C_VEL
LIN {X 0,Y 460.023,Z 433.751,A -85,B 0,C 180,E1 -8398.045,E2 -8398.045} C_VEL
LIN {X 0,Y 461.794,Z 405.487,A -85,B 0,C 180,E1 -8401.159,E2 -8401.159} C_VEL
LIN {X 0,Y 461.599,Z 402.596,A -85,B 0,C 180,E1 -8401.502,E2 -8401.502} C_VEL
LIN {X 0,Y 456.1,Z 383.518,A -85,B 0,C 180,E1 -8404.083,E2 -8404.083} C_VEL
LIN {X 0,Y 453.505,Z 374.884,A -85,B 0,C 180,E1 -8405.324,E2 -8405.324} C_VEL
LIN {X 0,Y 453.43,Z 374.631,A -85,B 0,C 180,E1 -8406.295,E2 -8406.295} C_VEL
LIN {X 0,Y 453.431,Z 374.629,A -85,B 0,C 180,E1 -8409.453,E2 -8409.453} C_VEL
LIN {X 0,Y 453.436,Z 374.63,A -85,B 0,C 180,E1 -8411.929,E2 -8411.929} C_VEL
LIN {X 0,Y 453.464,Z 374.622,A -85,B 0,C 180,E1 -8415.471,E2 -8415.471} C_VEL
LIN {X 0,Y 453.457,Z 374.615,A -85,B 0,C 180,E1 -8419.387,E2 -8419.387} C_VEL
LIN {X 0,Y 453.421,Z 374.617,A -85,B 0,C 180,E1 -8422.807,E2 -8422.807} C_VEL
LIN {X 0,Y 453.451,Z 374.604,A -85,B 0,C 180,E1 -8426.085,E2 -8426.085} C_VEL
LIN {X 0,Y 453.459,Z 374.622,A -85,B 0,C 180,E1 -8429.239,E2 -8429.239} C_VEL
LIN {X 0,Y 453.46,Z 374.624,A -85,B 0,C 180,E1 -8432.293,E2 -8432.293} C_VEL
LIN {X 0,Y 453.457,Z 374.613,A -85,B 0,C 180,E1 -8435.262,E2 -8435.262} C_VEL
LIN {X 0,Y 453.465,Z 374.624,A -85,B 0,C 180,E1 -8438.415,E2 -8438.415} C_VEL
LIN {X 0,Y 453.507,Z 374.616,A -85,B 0,C 180,E1 -8441.008,E2 -8441.008} C_VEL
LIN {X 0,Y 453.502,Z 374.61,A -85,B 0,C 180,E1 -8444.725,E2 -8444.725} C_VEL
LIN {X 0,Y 453.539,Z 374.617,A -85,B 0,C 180,E1 -8448.379,E2 -8448.379} C_VEL
LIN {X 0,Y 453.544,Z 374.608,A -85,B 0,C 180,E1 -8451.086,E2 -8451.086} C_VEL
LIN {X 0,Y 453.611,Z 374.602,A -85,B 0,C 180,E1 -8453.774,E2 -8453.774} C_VEL
LIN {X 0,Y 453.696,Z 374.591,A -85,B 0,C 180,E1 -8457.337,E2 -8457.337} C_VEL
LIN {X 0,Y 453.729,Z 374.588,A -85,B 0,C 180,E1 -8460,E2 -8460} C_VEL
LIN {X 0,Y 453.692,Z 374.593,A -85,B 0,C 180,E1 -8462.664,E2 -8462.664} C_VEL
LIN {X 0,Y 453.638,Z 374.595,A -85,B 0,C 180,E1 -8466.226,E2 -8466.226} C_VEL
LIN {X 0,Y 453.558,Z 374.613,A -85,B 0,C 180,E1 -8468.914,E2 -8468.914} C_VEL
LIN {X 0,Y 453.548,Z 374.604,A -85,B 0,C 180,E1 -8472.529,E2 -8472.529} C_VEL
LIN {X 0,Y 453.529,Z 374.609,A -85,B 0,C 180,E1 -8476.197,E2 -8476.197} C_VEL
LIN {X 0,Y 453.501,Z 374.618,A -85,B 0,C 180,E1 -8479.04,E2 -8479.04} C_VEL
LIN {X 0,Y 453.461,Z 374.616,A -85,B 0,C 180,E1 -8481.837,E2 -8481.837} C_VEL
LIN {X 0,Y 453.449,Z 374.622,A -85,B 0,C 180,E1 -8484.738,E2 -8484.738} C_VEL
LIN {X 0,Y 453.447,Z 374.625,A -85,B 0,C 180,E1 -8487.943,E2 -8487.943} C_VEL
LIN {X 0,Y 453.439,Z 374.631,A -85,B 0,C 180,E1 -8490.762,E2 -8490.762} C_VEL
LIN {X 0,Y 453.453,Z 374.625,A -85,B 0,C 180,E1 -8493.915,E2 -8493.915} C_VEL
LIN {X 0,Y 453.426,Z 374.608,A -85,B 0,C 180,E1 -8497.192,E2 -8497.192} C_VEL
LIN {X 0,Y 453.458,Z 374.627,A -85,B 0,C 180,E1 -8500.613,E2 -8500.613} C_VEL
LIN {X 0,Y 453.464,Z 374.625,A -85,B 0,C 180,E1 -8504.529,E2 -8504.529} C_VEL
LIN {X 0,Y 453.431,Z 374.629,A -85,B 0,C 180,E1 -8508.206,E2 -8508.206} C_VEL
LIN {X 0,Y 453.428,Z 374.621,A -85,B 0,C 180,E1 -8510.804,E2 -8510.804} C_VEL
LIN {X 0,Y 453.43,Z 374.787,A -85,B 0,C 180,E1 -8513.572,E2 -8513.572} C_VEL
LIN {X 0,Y 454.29,Z 377.421,A -85,B 0,C 180,E1 -8513.996,E2 -8513.996} C_VEL
LIN {X 0,Y 458.9,Z 392.206,A -85,B 0,C 180,E1 -8516.09,E2 -8516.09} C_VEL
LIN {X 0,Y 462.34,Z 405.287,A -85,B 0,C 180,E1 -8517.859,E2 -8517.859} C_VEL
LIN {X 0,Y 460.904,Z 433.41,A -85,B 0,C 180,E1 -8521.046,E2 -8521.046} C_VEL
LIN {X 0,Y 459.533,Z 464.735,A -85,B 0,C 180,E1 -8524.467,E2 -8524.467} C_VEL
LIN {X 0,Y 459.282,Z 472.256,A -85,B 0,C 180,E1 -8525.222,E2 -8525.222} C_VEL
LIN {X 0,Y 462.994,Z 494.952,A -85,B 0,C 180,E1 -8525.825,E2 -8525.825} C_VEL
LIN {X 0,Y 462.349,Z 543.721,A -85,B 0,C 180,E1 -8526.602,E2 -8526.602} C_VEL
LIN {X 0,Y 461.693,Z 549.569,A -85,B 0,C 180,E1 -8526.664,E2 -8526.664} C_VEL
LIN {X 0,Y 456.115,Z 568.62,A -85,B 0,C 180,E1 -8526.684,E2 -8526.684} C_VEL
LIN {X 0,Y 455.399,Z 574.472,A -85,B 0,C 180,E1 -8526.745,E2 -8526.745} C_VEL
LIN {X 0,Y 454.39,Z 640.332,A -85,B 0,C 180,E1 -8527.824,E2 -8527.824} C_VEL
LIN {X 0,Y 453.943,Z 655.846,A -85,B 0,C 180,E1 -8528.247,E2 -8528.247} C_VEL
LIN {X 0,Y 453.238,Z 669.953,A -85,B 0,C 180,E1 -8528.796,E2 -8528.796} C_VEL
LIN {X 0,Y 452.384,Z 684.378,A -85,B 0,C 180,E1 -8529.542,E2 -8529.542} C_VEL
LIN {X 0,Y 451.401,Z 698.142,A -85,B 0,C 180,E1 -8530.445,E2 -8530.445} C_VEL
LIN {X 0,Y 450.357,Z 712.046,A -85,B 0,C 180,E1 -8531.58,E2 -8531.58} C_VEL
LIN {X 0,Y 449.376,Z 724.594,A -85,B 0,C 180,E1 -8532.832,E2 -8532.832} C_VEL
LIN {X 0,Y 448.473,Z 735.117,A -85,B 0,C 180,E1 -8534.085,E2 -8534.085} C_VEL
LIN {X 0,Y 447.682,Z 744.869,A -85,B 0,C 180,E1 -8535.454,E2 -8535.454} C_VEL
LIN {X 0,Y 447.01,Z 753.438,A -85,B 0,C 180,E1 -8536.87,E2 -8536.87} C_VEL
LIN {X 0,Y 446.436,Z 762.359,A -85,B 0,C 180,E1 -8538.653,E2 -8538.653} C_VEL
LIN {X 0,Y 445.903,Z 769.771,A -85,B 0,C 180,E1 -8540.476,E2 -8540.476} C_VEL
LIN {X 0,Y 445.622,Z 775.659,A -85,B 0,C 180,E1 -8542.298,E2 -8542.298} C_VEL
LIN {X 0,Y 445.459,Z 779.213,A -85,B 0,C 180,E1 -8543.696,E2 -8543.696} C_VEL
LIN {X 0,Y 445.376,Z 782.673,A -85,B 0,C 180,E1 -8545.476,E2 -8545.476} C_VEL
LIN {X 0,Y 445.391,Z 785.015,A -85,B 0,C 180,E1 -8547.288,E2 -8547.288} C_VEL
LIN {X 0,Y 445.312,Z 786.209,A -85,B 0,C 180,E1 -8549.097,E2 -8549.097} C_VEL
LIN {X 0,Y 445.313,Z 786.225,A -85,B 0,C 180,E1 -8550.906,E2 -8550.906} C_VEL
LIN {X 0,Y 445.392,Z 785.096,A -85,B 0,C 180,E1 -8552.715,E2 -8552.715} C_VEL
LIN {X 0,Y 445.375,Z 782.817,A -85,B 0,C 180,E1 -8554.527,E2 -8554.527} C_VEL
LIN {X 0,Y 445.53,Z 779.229,A -85,B 0,C 180,E1 -8556.387,E2 -8556.387} C_VEL
LIN {X 0,Y 445.683,Z 774.571,A -85,B 0,C 180,E1 -8558.16,E2 -8558.16} C_VEL
LIN {X 0,Y 445.958,Z 768.402,A -85,B 0,C 180,E1 -8559.984,E2 -8559.984} C_VEL
LIN {X 0,Y 446.549,Z 760.643,A -85,B 0,C 180,E1 -8561.807,E2 -8561.807} C_VEL
LIN {X 0,Y 447.054,Z 752.501,A -85,B 0,C 180,E1 -8563.386,E2 -8563.386} C_VEL
LIN {X 0,Y 447.875,Z 742.402,A -85,B 0,C 180,E1 -8565.007,E2 -8565.007} C_VEL
LIN {X 0,Y 448.712,Z 732.232,A -85,B 0,C 180,E1 -8566.376,E2 -8566.376} C_VEL
LIN {X 0,Y 449.714,Z 720.473,A -85,B 0,C 180,E1 -8567.701,E2 -8567.701} C_VEL
LIN {X 0,Y 450.689,Z 707.893,A -85,B 0,C 180,E1 -8568.88,E2 -8568.88} C_VEL
LIN {X 0,Y 451.643,Z 694.643,A -85,B 0,C 180,E1 -8569.902,E2 -8569.902} C_VEL
LIN {X 0,Y 452.625,Z 681.005,A -85,B 0,C 180,E1 -8570.746,E2 -8570.746} C_VEL
LIN {X 0,Y 453.383,Z 666.874,A -85,B 0,C 180,E1 -8571.436,E2 -8571.436} C_VEL
LIN {X 0,Y 454.104,Z 651.59,A -85,B 0,C 180,E1 -8571.985,E2 -8571.985} C_VEL
LIN {X 0,Y 454.538,Z 636.238,A -85,B 0,C 180,E1 -8572.351,E2 -8572.351} C_VEL
LIN {X 0,Y 456.504,Z 496.077,A -85,B 0,C 180,E1 -8574.614,E2 -8574.614} C_VEL
LIN {X 0,Y 452.634,Z 471.887,A -85,B 0,C 180,E1 -8575.278,E2 -8575.278} C_VEL
LIN {X 0,Y 453.594,Z 448.324,A -85,B 0,C 180,E1 -8577.802,E2 -8577.802} C_VEL
LIN {X 0,Y 455.077,Z 419.756,A -85,B 0,C 180,E1 -8581.027,E2 -8581.027} C_VEL
LIN {X 0,Y 455.723,Z 407.481,A -85,B 0,C 180,E1 -8582.434,E2 -8582.434} C_VEL
LIN {X 0,Y 452.606,Z 395.667,A -85,B 0,C 180,E1 -8584.068,E2 -8584.068} C_VEL
LIN {X 0,Y 447.522,Z 379.339,A -85,B 0,C 180,E1 -8586.405,E2 -8586.405} C_VEL
LIN {X 0,Y 446.389,Z 375.67,A -85,B 0,C 180,E1 -8586.994,E2 -8586.994} C_VEL
LIN {X 0,Y 446.39,Z 375.506,A -85,B 0,C 180,E1 -8590.205,E2 -8590.205} C_VEL
LIN {X 0,Y 446.381,Z 375.509,A -85,B 0,C 180,E1 -8593.594,E2 -8593.594} C_VEL
LIN {X 0,Y 446.377,Z 375.498,A -85,B 0,C 180,E1 -8596.408,E2 -8596.408} C_VEL
LIN {X 0,Y 446.391,Z 375.487,A -85,B 0,C 180,E1 -8599.796,E2 -8599.796} C_VEL
LIN {X 0,Y 446.395,Z 375.502,A -85,B 0,C 180,E1 -8603.254,E2 -8603.254} C_VEL
LIN {X 0,Y 446.429,Z 375.488,A -85,B 0,C 180,E1 -8606.551,E2 -8606.551} C_VEL
LIN {X 0,Y 446.431,Z 375.499,A -85,B 0,C 180,E1 -8609.981,E2 -8609.981} C_VEL
LIN {X 0,Y 446.388,Z 375.507,A -85,B 0,C 180,E1 -8612.833,E2 -8612.833} C_VEL
LIN {X 0,Y 446.473,Z 375.496,A -85,B 0,C 180,E1 -8616.334,E2 -8616.334} C_VEL
LIN {X 0,Y 446.526,Z 375.716,A -85,B 0,C 180,E1 -8616.859,E2 -8616.859} C_VEL
LIN {X 0,Y 448.352,Z 384.031,A -85,B 0,C 180,E1 -8618.478,E2 -8618.478} C_VEL
LIN {X 0,Y 452.749,Z 396.393,A -85,B 0,C 180,E1 -8618.94,E2 -8618.94} C_VEL
LIN {X 0,Y 453.545,Z 400.984,A -85,B 0,C 180,E1 -8619.067,E2 -8619.067} C_VEL
LIN {X 0,Y 451.62,Z 509.139,A -85,B 0,C 180,E1 -8621.073,E2 -8621.073} C_VEL
LIN {X 0,Y 451.359,Z 527.95,A -85,B 0,C 180,E1 -8621.474,E2 -8621.474} C_VEL
LIN {X 0,Y 451.1,Z 542.943,A -85,B 0,C 180,E1 -8621.986,E2 -8621.986} C_VEL
LIN {X 0,Y 450.738,Z 557.142,A -85,B 0,C 180,E1 -8622.666,E2 -8622.666} C_VEL
LIN {X 0,Y 450.176,Z 569.839,A -85,B 0,C 180,E1 -8623.446,E2 -8623.446} C_VEL
LIN {X 0,Y 449.713,Z 581.785,A -85,B 0,C 180,E1 -8624.361,E2 -8624.361} C_VEL
LIN {X 0,Y 449.08,Z 593.972,A -85,B 0,C 180,E1 -8625.499,E2 -8625.499} C_VEL
LIN {X 0,Y 448.568,Z 604.075,A -85,B 0,C 180,E1 -8626.638,E2 -8626.638} C_VEL
LIN {X 0,Y 447.99,Z 614.16,A -85,B 0,C 180,E1 -8628.003,E2 -8628.003} C_VEL
LIN {X 0,Y 447.531,Z 622.52,A -85,B 0,C 180,E1 -8629.367,E2 -8629.367} C_VEL
LIN {X 0,Y 447.162,Z 630.529,A -85,B 0,C 180,E1 -8630.957,E2 -8630.957} C_VEL
LIN {X 0,Y 446.85,Z 635.861,A -85,B 0,C 180,E1 -8632.25,E2 -8632.25} C_VEL
LIN {X 0,Y 446.632,Z 640.689,A -85,B 0,C 180,E1 -8633.676,E2 -8633.676} C_VEL
LIN {X 0,Y 446.509,Z 644.36,A -85,B 0,C 180,E1 -8635.034,E2 -8635.034} C_VEL
LIN {X 0,Y 446.292,Z 647.13,A -85,B 0,C 180,E1 -8636.388,E2 -8636.388} C_VEL
LIN {X 0,Y 446.39,Z 648.521,A -85,B 0,C 180,E1 -8637.293,E2 -8637.293} C_VEL
LIN {X 0,Y 446.342,Z 650.308,A -85,B 0,C 180,E1 -8639.098,E2 -8639.098} C_VEL
LIN {X 0,Y 446.353,Z 650.728,A -85,B 0,C 180,E1 -8640.902,E2 -8640.902} C_VEL
LIN {X 0,Y 446.527,Z 649.736,A -85,B 0,C 180,E1 -8642.706,E2 -8642.706} C_VEL
LIN {X 0,Y 446.601,Z 647.358,A -85,B 0,C 180,E1 -8644.513,E2 -8644.513} C_VEL
LIN {X 0,Y 446.987,Z 643.478,A -85,B 0,C 180,E1 -8646.319,E2 -8646.319} C_VEL
LIN {X 0,Y 447.391,Z 638.02,A -85,B 0,C 180,E1 -8648.128,E2 -8648.128} C_VEL
LIN {X 0,Y 447.735,Z 632.769,A -85,B 0,C 180,E1 -8649.486,E2 -8649.486} C_VEL
LIN {X 0,Y 448.308,Z 625.185,A -85,B 0,C 180,E1 -8651.072,E2 -8651.072} C_VEL
LIN {X 0,Y 448.901,Z 617.187,A -85,B 0,C 180,E1 -8652.431,E2 -8652.431} C_VEL
LIN {X 0,Y 449.562,Z 607.403,A -85,B 0,C 180,E1 -8653.805,E2 -8653.805} C_VEL
LIN {X 0,Y 450.262,Z 596.667,A -85,B 0,C 180,E1 -8655.04,E2 -8655.04} C_VEL
LIN {X 0,Y 450.916,Z 584.586,A -85,B 0,C 180,E1 -8656.177,E2 -8656.177} C_VEL
LIN {X 0,Y 451.451,Z 572.736,A -85,B 0,C 180,E1 -8657.088,E2 -8657.088} C_VEL
LIN {X 0,Y 452.058,Z 558.695,A -85,B 0,C 180,E1 -8657.94,E2 -8657.94} C_VEL
LIN {X 0,Y 452.519,Z 544.976,A -85,B 0,C 180,E1 -8658.573,E2 -8658.573} C_VEL
LIN {X 0,Y 452.708,Z 530.57,A -85,B 0,C 180,E1 -8659.056,E2 -8659.056} C_VEL
LIN {X 0,Y 454.896,Z 453.347,A -85,B 0,C 180,E1 -8660.755,E2 -8660.755} C_VEL
LIN {X 0,Y 456.742,Z 404.095,A -85,B 0,C 180,E1 -8661.893,E2 -8661.893} C_VEL
LIN {X 0,Y 451.708,Z 394.183,A -85,B 0,C 180,E1 -8662.58,E2 -8662.58} C_VEL
LIN {X 0,Y 449.409,Z 385.158,A -85,B 0,C 180,E1 -8664.976,E2 -8664.976} C_VEL
LIN {X 0,Y 446.653,Z 376.266,A -85,B 0,C 180,E1 -8667.657,E2 -8667.657} C_VEL
LIN {X 0,Y 446.521,Z 375.563,A -85,B 0,C 180,E1 -8667.921,E2 -8667.921} C_VEL
LIN {X 0,Y 446.421,Z 375.505,A -85,B 0,C 180,E1 -8671.3,E2 -8671.3} C_VEL
LIN {X 0,Y 446.433,Z 375.503,A -85,B 0,C 180,E1 -8674.523,E2 -8674.523} C_VEL
LIN {X 0,Y 446.415,Z 375.505,A -85,B 0,C 180,E1 -8678.078,E2 -8678.078} C_VEL
LIN {X 0,Y 446.426,Z 375.503,A -85,B 0,C 180,E1 -8680.916,E2 -8680.916} C_VEL
LIN {X 0,Y 446.402,Z 375.507,A -85,B 0,C 180,E1 -8683.846,E2 -8683.846} C_VEL
LIN {X 0,Y 446.391,Z 375.509,A -85,B 0,C 180,E1 -8686.404,E2 -8686.404} C_VEL
LIN {X 0,Y 446.4,Z 375.508,A -85,B 0,C 180,E1 -8689.796,E2 -8689.796} C_VEL
LIN {X 0,Y 446.417,Z 375.679,A -85,B 0,C 180,E1 -8692.477,E2 -8692.477} C_VEL
LIN {X 0,Y 448.969,Z 382.676,A -85,B 0,C 180,E1 -8694.103,E2 -8694.103} C_VEL
LIN {X 0,Y 451.855,Z 391.148,A -85,B 0,C 180,E1 -8695.779,E2 -8695.779} C_VEL
LIN {X 0,Y 454.6,Z 401.151,A -85,B 0,C 180,E1 -8697.504,E2 -8697.504} C_VEL
LIN {X 0,Y 455.746,Z 406.8,A -85,B 0,C 180,E1 -8698.377,E2 -8698.377} C_VEL
LIN {X 0,Y 453.385,Z 431.768,A -85,B 0,C 180,E1 -8701.418,E2 -8701.418} C_VEL
LIN {X 0,Y 451.547,Z 457.619,A -85,B 0,C 180,E1 -8704.416,E2 -8704.416} C_VEL
LIN {X 0,Y 451.483,Z 459.418,A -85,B 0,C 180,E1 -8704.588,E2 -8704.588} C_VEL
LIN {X 0,Y 453.983,Z 478.247,A -85,B 0,C 180,E1 -8705.207,E2 -8705.207} C_VEL
LIN {X 0,Y 455.738,Z 494.504,A -85,B 0,C 180,E1 -8705.632,E2 -8705.632} C_VEL
LIN {X 0,Y 453.847,Z 638.948,A -85,B 0,C 180,E1 -8707.972,E2 -8707.972} C_VEL
LIN {X 0,Y 453.433,Z 653.54,A -85,B 0,C 180,E1 -8708.351,E2 -8708.351} C_VEL
LIN {X 0,Y 452.779,Z 667.72,A -85,B 0,C 180,E1 -8708.881,E2 -8708.881} C_VEL
LIN {X 0,Y 451.964,Z 682.709,A -85,B 0,C 180,E1 -8709.638,E2 -8709.638} C_VEL
LIN {X 0,Y 451.067,Z 696.678,A -85,B 0,C 180,E1 -8710.545,E2 -8710.545} C_VEL
LIN {X 0,Y 450.132,Z 709.418,A -85,B 0,C 180,E1 -8711.568,E2 -8711.568} C_VEL
LIN {X 0,Y 449.147,Z 722.012,A -85,B 0,C 180,E1 -8712.794,E2 -8712.794} C_VEL
LIN {X 0,Y 448.291,Z 732.973,A -85,B 0,C 180,E1 -8714.075,E2 -8714.075} C_VEL
LIN {X 0,Y 447.582,Z 742.864,A -85,B 0,C 180,E1 -8715.448,E2 -8715.448} C_VEL
LIN {X 0,Y 446.815,Z 752.517,A -85,B 0,C 180,E1 -8717.046,E2 -8717.046} C_VEL
LIN {X 0,Y 446.356,Z 760.545,A -85,B 0,C 180,E1 -8718.648,E2 -8718.648} C_VEL
LIN {X 0,Y 445.891,Z 768.01,A -85,B 0,C 180,E1 -8720.473,E2 -8720.473} C_VEL
LIN {X 0,Y 445.659,Z 773.925,A -85,B 0,C 180,E1 -8722.295,E2 -8722.295} C_VEL
LIN {X 0,Y 445.577,Z 777.42,A -85,B 0,C 180,E1 -8723.66,E2 -8723.66} C_VEL
LIN {X 0,Y 445.456,Z 780.972,A -85,B 0,C 180,E1 -8725.474,E2 -8725.474} C_VEL
LIN {X 0,Y 445.483,Z 783.306,A -85,B 0,C 180,E1 -8727.286,E2 -8727.286} C_VEL
LIN {X 0,Y 445.385,Z 784.478,A -85,B 0,C 180,E1 -8729.094,E2 -8729.094} C_VEL
LIN {X 0,Y 445.385,Z 784.478,A -85,B 0,C 180,E1 -8730.903,E2 -8730.903} C_VEL
LIN {X 0,Y 445.486,Z 783.303,A -85,B 0,C 180,E1 -8732.711,E2 -8732.711} C_VEL
LIN {X 0,Y 445.44,Z 780.971,A -85,B 0,C 180,E1 -8734.523,E2 -8734.523} C_VEL
LIN {X 0,Y 445.526,Z 777.319,A -85,B 0,C 180,E1 -8736.384,E2 -8736.384} C_VEL
LIN {X 0,Y 445.704,Z 772.577,A -85,B 0,C 180,E1 -8738.157,E2 -8738.157} C_VEL
LIN {X 0,Y 445.954,Z 766.291,A -85,B 0,C 180,E1 -8739.981,E2 -8739.981} C_VEL
LIN {X 0,Y 446.433,Z 759.499,A -85,B 0,C 180,E1 -8741.577,E2 -8741.577} C_VEL
LIN {X 0,Y 446.892,Z 751.287,A -85,B 0,C 180,E1 -8743.18,E2 -8743.18} C_VEL
LIN {X 0,Y 447.611,Z 741.374,A -85,B 0,C 180,E1 -8744.78,E2 -8744.78} C_VEL
